	// **********************************************************
	// *                 MANAGEMENT TRANSITION                  *
	// **********************************************************
	
	// Transition from Stop to WarmUp
	
	IF "SM1".xBattOpenSt AND NOT "SM1".xStopAutomaintCmd        //Whit battery open and not automaintenance go to warmup state
	THEN
	    "SM1".xT81 := True;
	END_IF;
	
	// Reset Transition
	
	"SM1".xT32   := False;
	"SM1".xT43   := False;
	"SM1".xT52   := False;
	"SM1".xT72   := False;
	
END_FUNCTION

FUNCTION "SM1_S9_Fault" : Void
{ S7_Optimized_Access := 'TRUE' }
VERSION : 0.1

BEGIN
	// **********************************************************
	// *                   MANAGEMENT ACTION                    *
	// **********************************************************
	
	REGION State Machine Status
	    
	    "SM1".xSsBootSt      := False;
	    "SM1".xSsWarmUpSt    := False;
	    "SM1".xSsReadySt     := False;
	    "SM1".xSsStandBySt   := False;
	    "SM1".xSsRunSt       := False;
	    "SM1".xSsTestSt      := False;
	    "SM1".xSsAutoMaintSt := False;
	    "SM1".xSsStopSt      := False;
	    "SM1".xSsFaultSt     := True;
	    
	    "SM1".iCountSS := 9;
	    
	END_REGION
	
	"SM1".xPCSrunCmd := False;      //In fault state send stop command to the PCS
	
	REGION PCS enable Off
	    
	    IF "SM1".xPCSreadySt        //When the PCS are in ready take out the enable command to the PCS
	    THEN
	        "SM1".xPCSenbCmd := False;
	    END_IF;
	END_REGION
	
	REGION Command Open RMU and Battery
	    
	    IF "SM1".xPCSstopSt AND NOT "SM1".xVacPCS       //When we go in fault state have a possibility who the medium voltage is off
	    THEN
	        "SM1".xMVbreakerOpenCmd := True;        //If the medium voltage is off we need to open a MV breaker because otherwise after giving the open command to the battery,
	                                                //the PCS would switch off AND in this CASE you could NOT close the MV breaker anymore
	        IF "SM1".xMVbreakerOpenSt       //When the MV breaker are opened semd a open command to the battery
	        THEN
	            "SM1".xBattCloseCmd := False;
	        END_IF;
	    END_IF;
	    
	END_REGION
	
	REGION Command Open Battery
	    
	    IF "SM1".xPCSstopSt AND "SM1".xVacPCS       //If the medium voltage is on and PCS stopped send a open command to the battery
	    THEN
	        "SM1".xBattCloseCmd := False;
	    END_IF;
	    
	END_REGION
	
	
	// **********************************************************
	// *                 MANAGEMENT TRANSITION                  *
	// **********************************************************
	
	// Transition from Alarm to WarmUp
	
	IF NOT "SM1".xFltSt AND "SM1".xBattOpenSt       //Without faults and battery open return in warmup state
	THEN
	    "SM1".xT91 := True;
	    "SM1".xMVbreakerOpenCmd := False;
	END_IF;
	
	// Reset Transition
	
	"SM1".xT22   := False;
	"SM1".xT33   := False;
	"SM1".xT44   := False;
	"SM1".xT53   := False;
	"SM1".xT62   := False;
	"SM1".xT73   := False;
	
END_FUNCTION

FUNCTION "SM2_S1_Boot" : Void
{ S7_Optimized_Access := 'TRUE' }
VERSION : 0.1
   VAR_TEMP 
      xBoot_Ok : Bool;
      iT1 : S5Time;
   END_VAR


BEGIN
	// **********************************************************
	// *                   MANAGEMENT ACTION                    *
	// **********************************************************
	
	REGION State Machine Status
	    
	    "SM2".xSsBootSt      := True;
	    "SM2".xSsWarmUpSt    := False;
	    "SM2".xSsReadySt     := False;
	    "SM2".xSsStandBySt   := False;
	    "SM2".xSsRunSt       := False;
	    "SM2".xSsTestSt      := False;
	    "SM2".xSsAutoMaintSt := False;
	    "SM2".xSsStopSt      := False;
	    "SM2".xSsFaultSt     := False;
	    
	    "SM2".iCountSS := 1;
	    
	END_REGION
	
	REGION Wait PLC Status From Off to On
	    
	// When the PLC switch to Run after 5sec "xBootSt = True" and the transition "T1 = True"
	    
	#iT1 := S_ODT(
	    T_NO := 1,
	    S := "SM2".xRunPlcSt,
	    TV := S5T#5s,
	    Q => "SM2".xBootSt);
	END_REGION
	
	// **********************************************************
	// *                 MANAGEMENT TRANSITION                  *
	// **********************************************************
	
	// Transition from Boot to WarmUp
	
	IF "SM2".xBootSt
	THEN
	    "SM2".xT11 := True;
	    "SM2".xBootSt := False;
	END_IF;
	
END_FUNCTION

FUNCTION "SM2_S2_WarmUp" : Void
{ S7_Optimized_Access := 'TRUE' }
VERSION : 0.1
   VAR_TEMP 
      xWarmUpSt : Bool;
   END_VAR


BEGIN
	// **********************************************************
	// *                   MANAGEMENT ACTION                    *
	// **********************************************************
	
	REGION State Machine Status
	    
	    "SM2".xSsBootSt      := False;
	    "SM2".xSsWarmUpSt    := True;
	    "SM2".xSsReadySt     := False;
	    "SM2".xSsStandBySt   := False;
	    "SM2".xSsRunSt       := False;
	    "SM2".xSsTestSt      := False;
	    "SM2".xSsAutoMaintSt := False;
	    "SM2".xSsStopSt      := False;
	    "SM2".xSsFaultSt     := False;
	    
	    "SM2".iCountSS       := 2;
	    
	END_REGION
	
	REGION Activation
	    
	    "SM2".xCommCmd   := True;    //Enable all communication on the Power Island
	    "SM2".xAuxCmd    := True;    //Enable all auxiliary equipment on the Power Island
	    
	END_REGION
	
	REGION Activation Active
	    
	    IF "SM2".xAuxSt AND "SM2".xCommSt     //Check the feedback of communication and auxiliary on the Power Island
	    THEN
	        #xWarmUpSt := True;
	
	    END_IF;
	    
	END_REGION
	
	
	// **********************************************************
	// *                 MANAGEMENT TRANSITION                  *
	// **********************************************************
	
	// Transition from WarmUp to Ready
	
	IF #xWarmUpSt
	THEN
	    "SM2".xT21 := True;
	    #xWarmUpSt := False;
	END_IF;
	
	// Transition from WarmUp to Fault
	
	IF "SM2".xFltSt
	THEN
	    "SM2".xT22 := True;
	END_IF;
	
	// Reset Transition
	
	"SM2".xT11   := False;
	"SM2".xT81   := False;
	"SM2".xT91   := False;
	
END_FUNCTION

FUNCTION "SM2_S3_Ready" : Void
{ S7_Optimized_Access := 'TRUE' }
VERSION : 0.1
   VAR_TEMP 
      xSSysReadySt : Bool;
   END_VAR


BEGIN
	// **********************************************************
	// *                   MANAGEMENT ACTION                    *
	// **********************************************************
	
	REGION State Machine Status
	    
	    "SM2".xSsBootSt      := False;
	    "SM2".xSsWarmUpSt    := False;
	    "SM2".xSsReadySt     := True;
	    "SM2".xSsStandBySt   := False;
	    "SM2".xSsRunSt       := False;
	    "SM2".xSsTestSt      := False;
	    "SM2".xSsAutoMaintSt := False;
	    "SM2".xSsStopSt      := False;
	    "SM2".xSsFaultSt     := False;
	        
	    "SM2".iCountSS := 3;
	    
	END_REGION
	
	REGION Ready Condition
	    
	    IF "SM2".xReadyCondSt AND "SM2".xEnbSSysSt      //With ready condition and Subsystem enabled from HMI the subsystem is ready
	    THEN
	        #xSSysReadySt := True;
	    END_IF;
	    
	END_REGION
	
	REGION Command Battery Close
	    
	    IF #xSSysReadySt AND ("SM2".xStandByCmd OR "SM2".xRunCmd)       //With subsystem ready and standby or run command send close command to the battery
	    THEN
	        "SM2".xBattCloseCmd := True;
	    END_IF;
	    
	END_REGION
	
	REGION Command Enable PCS
	    
	    IF "SM2".xBattCloseSt AND "SM2".xMVbreakerCloseSt       //When the battery are closed and MV circuit breaker close send enable command to the PCS
	    THEN
	        "SM2".xPCSenbCmd := True;
	    END_IF;
	END_REGION
	
	
	// **********************************************************
	// *                 MANAGEMENT TRANSITION                  *
	// **********************************************************
	
	// Transition from Ready to StandBy
	
	IF "SM2".xBattCloseSt AND "SM2".xPCSreadySt     //With battery closed and PCS in ready condition go on standby state
	THEN
	    "SM2".xT31 := True;
	    #xSSysReadySt := False;
	END_IF;
	
	// Transition from Ready to Stop
	
	IF "SM2".xStopCmd AND False     //From ready status never go in stop state
	THEN
	    "SM2".xT32 := True;
	END_IF;
	
	// Transition from Ready to Fault
	
	IF "SM2".xFltSt     //With subsystem in fault go to the fault state
	THEN
	    "SM2".xT33 := True;
	END_IF;
	
	// Transition from Ready to Test
	
	IF "SM2".xTestCmd       //With test command from HMI go to the test state
	THEN
	    "SM2".xT34 := True;
	END_IF;
	
	// Reset Transition
	
	"SM2".xT21   := False;
	"SM2".xT61   := False;
	
END_FUNCTION

FUNCTION "SM2_S4_StandBy" : Void
{ S7_Optimized_Access := 'TRUE' }
VERSION : 0.1

BEGIN
	// **********************************************************
	// *                   MANAGEMENT ACTION                    *
	// **********************************************************
	
	REGION State Machine Status
	    
	    "SM2".xSsBootSt      := False;
	    "SM2".xSsWarmUpSt    := False;
	    "SM2".xSsReadySt     := False;
	    "SM2".xSsStandBySt   := True;
	    "SM2".xSsRunSt       := False;
	    "SM2".xSsTestSt      := False;
	    "SM2".xSsAutoMaintSt := False;
	    "SM2".xSsStopSt      := False;
	    "SM2".xSsFaultSt     := False;
	    
	    "SM2".iCountSS := 4;
	    
	END_REGION
	
	REGION Run Command
	    
	    IF "SM2".xRunCmd        //With run command send run command to the PCS
	    THEN
	        "SM2".xPCSrunCmd := True;
	    END_IF;
	    
	END_REGION
	
	
	// **********************************************************
	// *                 MANAGEMENT TRANSITION                  *
	// **********************************************************
	
	// Transition from StandBy to Run
	
	IF "SM2".xPCSrunSt AND "SM2".xRunCmd        //With PCS in run and the command on go to run state
	THEN
	    "SM2".xT41 := True;
	END_IF;
	
	// Transition from StandBy to AutoMaint
	
	IF "SM2".xAutomaintCmd      //With automaintenance command go to automaintenance state
	THEN
	    "SM2".xT42 := True;
	END_IF;
	
	// Transition from StandBy to Stop
	
	IF "SM2".xStopCmd OR NOT "SM2".xEnbSSysSt       //With stop command or subsystem not enabled go to stop state
	THEN
	    "SM2".xT43 := True;
	END_IF;
	
	// Transition from StandBy to Fault
	
	IF "SM2".xFltSt     //With subsystem in fault go to the fault state
	THEN
	    "SM2".xT44 := True;
	END_IF;
	
	// Reset Transition
	
	"SM2".xT31   := False;
	"SM2".xT51   := False;
	"SM2".xT71   := False;
	
END_FUNCTION

FUNCTION "SM2_S5_Run" : Void
{ S7_Optimized_Access := 'TRUE' }
VERSION : 0.1

BEGIN
	// **********************************************************
	// *                   MANAGEMENT ACTION                    *
	// **********************************************************
	
	REGION State Machine Status
	    
	    "SM2".xSsBootSt      := False;
	    "SM2".xSsWarmUpSt    := False;
	    "SM2".xSsReadySt     := False;
	    "SM2".xSsStandBySt   := False;
	    "SM2".xSsRunSt       := True;
	    "SM2".xSsTestSt      := False;
	    "SM2".xSsAutoMaintSt := False;
	    "SM2".xSsStopSt      := False;
	    "SM2".xSsFaultSt     := False;
	    
	    "SM2".iCountSS := 5;
	    
	END_REGION
	
	REGION StandBy Command
	    
	    IF "SM2".xStandByCmd        //With standby command send stop command to the PCS
	    THEN
	        "SM2".xPCSrunCmd := False;
	    END_IF;
	    
	END_REGION
	
	
	// **********************************************************
	// *                 MANAGEMENT TRANSITION                  *
	// **********************************************************
	
	// Transition from Run to StandBy
	
	IF "SM2".xStandByCmd AND "SM2".xPCSreadySt      //With standby command e PCS in ready return to standby state
	THEN
	    "SM2".xT51 := True;
	END_IF;
	
	// Transition from Run to Stop
	
	IF "SM2".xStopCmd OR NOT "SM2".xEnbSSysSt       //With stop command or subsystem not enabled go to stop state
	THEN
	    "SM2".xT52 := True;
	END_IF;
	
	// Transition from Run to Fault
	
	IF "SM2".xFltSt     //With subsystem in fault go to the fault state
	THEN
	    "SM2".xT53 := True;
	END_IF;
	
	// Reset Transition
	
	"SM2".xT41 := False;
	
END_FUNCTION

FUNCTION "SM2_S6_Test" : Void
{ S7_Optimized_Access := 'TRUE' }
VERSION : 0.1

BEGIN
	// **********************************************************
	// *                   MANAGEMENT ACTION                    *
	// **********************************************************
	
	REGION State Machine Status
	    
	    "SM2".xSsBootSt := False;
	    "SM2".xSsWarmUpSt := False;
	    "SM2".xSsReadySt := False;
	    "SM2".xSsStandBySt := False;
	    "SM2".xSsRunSt := False;
	    "SM2".xSsTestSt := True;
	    "SM2".xSsAutoMaintSt := False;
	    "SM2".xSsStopSt := False;
	    "SM2".xSsFaultSt := False;
	    
	    "SM2".iCountSS := 6;
	    
	END_REGION
	
	"SM2".xPCSrunCmd := False;      //All command in this state are not necessary but only for safety
	
	REGION PCS Enable Off
	    
	    IF "SM2".xPCSreadySt
	    THEN
	        "SM2".xPCSenbCmd := False;
	    END_IF;
	END_REGION
	
	REGION Command Open Battery
	    
	    IF "SM2".xPCSstopSt
	    THEN
	        "SM2".xBattCloseCmd := False;
	    END_IF;
	END_REGION
	
	
	// **********************************************************
	// *                 MANAGEMENT TRANSITION                  *
	// **********************************************************
	
	// Transition from Test to Ready
	
	IF NOT "SM2".xTestCmd       //Without test command return to ready state
	THEN
	    "SM2".xT61 := True;
	END_IF;
	
	// Transition from Test to Fault
	
	IF "SM2".xFltSt     //With subsystem in fault go to the fault state
	THEN
	    "SM2".xT62 := True;
	END_IF;
	
	// Reset Transition
	
	"SM2".xT34 := False;
	
END_FUNCTION

FUNCTION "SM2_S7_AutoMaint" : Void
{ S7_Optimized_Access := 'TRUE' }
VERSION : 0.1

BEGIN
	// **********************************************************
	// *                   MANAGEMENT ACTION                    *
	// **********************************************************
	
	REGION State Machine Status
	    
	    "SM2".xSsBootSt      := False;
	    "SM2".xSsWarmUpSt    := False;
	    "SM2".xSsReadySt     := False;
	    "SM2".xSsStandBySt   := False;
	    "SM2".xSsRunSt       := False;
	    "SM2".xSsTestSt      := False;
	    "SM2".xSsAutoMaintSt := True;
	    "SM2".xSsStopSt      := False;
	    "SM2".xSsFaultSt     := False;
	    
	    "SM2".iCountSS := 7;
	    
	END_REGION
	
	REGION Autocharge Bank
	    
	    "SM2".xPCSrunCmd := True;       //In automaintenance state send run command to the PCS
	    
	    IF "SM2".xPCSrunSt      //When PCS are in run read the active power reference from HMI
	    THEN
	        "SM2".rPacAutomRef := "HMI".rPacAutomRef;
	    END_IF;
	    
	END_REGION
	
	
	// **********************************************************
	// *                 MANAGEMENT TRANSITION                  *
	// **********************************************************
	
	// Transition from AutoMaint to StandBy
	
	IF "SM2".xAutomaintSt       //Without automaintenance command from battery return to standby state
	THEN
	    "SM2".xT71 := True;
	END_IF;
	
	// Transition from AutoMaint to Stop
	
	IF "SM2".xStopCmd       //With stop command go to stop state
	THEN
	    "SM2".xT72 := True;
	END_IF;
	
	// Transition from AutoMaint to Fault
	
	IF "SM2".xFltSt     //With subsystem in fault go to the fault state
	THEN
	    "SM2".xT73 := True;
	END_IF;
	
	// Reset Transition
	
	"SM2".xT42    := False;
	
END_FUNCTION

FUNCTION "SM2_S8_Stop" : Void
{ S7_Optimized_Access := 'TRUE' }
VERSION : 0.1

BEGIN
	// **********************************************************
	// *                   MANAGEMENT ACTION                    *
	// **********************************************************
	
	REGION State Machine Status
	    
	    "SM2".xSsBootSt      := False;
	    "SM2".xSsWarmUpSt    := False;
	    "SM2".xSsReadySt     := False;
	    "SM2".xSsStandBySt   := False;
	    "SM2".xSsRunSt       := False;
	    "SM2".xSsTestSt      := False;
	    "SM2".xSsAutoMaintSt := False;
	    "SM2".xSsStopSt      := True;
	    "SM2".xSsFaultSt     := False;
	    
	    "SM2".iCountSS := 8;
	    
	END_REGION
	
	"SM2".xPCSrunCmd := False;      //In stop state send stop command to the PCS
	
	REGION PCS Enable Off
	    
	    IF "SM2".xPCSreadySt        //When the PCS are in ready take out the enable command to the PCS
	    THEN
	        "SM2".xPCSenbCmd := False;
	    END_IF;
	END_REGION
	
	REGION Command Open Battery
	    
	    IF "SM2".xPCSstopSt     //When the PCS are in stop send open command to the battery
	    THEN
	        "SM2".xBattCloseCmd := False;
	    END_IF;
	END_REGION
	
	
	// **********************************************************
	// *                 MANAGEMENT TRANSITION                  *
	// **********************************************************
	
	// Transition from Stop to WarmUp
	
	IF "SM2".xBattOpenSt AND NOT "SM2".xStopAutomaintCmd        //Whit battery open and not automaintenance go to warmup state
	THEN
	    "SM2".xT81 := True;
	END_IF;
	
	// Reset Transition
	
	"SM2".xT32   := False;
	"SM2".xT43   := False;
	"SM2".xT52   := False;
	"SM2".xT72   := False;
	
END_FUNCTION

FUNCTION "SM2_S9_Fault" : Void
{ S7_Optimized_Access := 'TRUE' }
VERSION : 0.1

BEGIN
	// **********************************************************
	// *                   MANAGEMENT ACTION                    *
	// **********************************************************
	
	REGION State Machine Status
	    
	    "SM2".xSsBootSt      := False;
	    "SM2".xSsWarmUpSt    := False;
	    "SM2".xSsReadySt     := False;
	    "SM2".xSsStandBySt   := False;
	    "SM2".xSsRunSt       := False;
	    "SM2".xSsTestSt      := False;
	    "SM2".xSsAutoMaintSt := False;
	    "SM2".xSsStopSt      := False;
	    "SM2".xSsFaultSt     := True;
	    
	    "SM2".iCountSS := 9;
	    
	END_REGION
	
	"SM2".xPCSrunCmd := False;      //In fault state send stop command to the PCS
	
	REGION PCS Enable Off
	    
	    IF "SM2".xPCSreadySt        //When the PCS are in ready take out the enable command to the PCS
	    THEN
	        "SM2".xPCSenbCmd := False;
	    END_IF;
	END_REGION
	
	REGION Command Open RMU and Battery
	    
	    IF "SM2".xPCSstopSt AND NOT "SM2".xVacPCS       //When we go in fault state have a possibility who the medium voltage is off
	    THEN
	        "SM2".xMVbreakerOpenCmd := True;        //If the medium voltage is off we need to open a MV breaker because otherwise after giving the open command to the battery,
	                                                //the PCS would switch off AND in this CASE you could NOT close the MV breaker anymore        
	        IF "SM2".xMVbreakerOpenSt       //When the MV breaker are opened semd a open command to the battery
	        THEN
	            "SM2".xBattCloseCmd := False;
	        END_IF;
	    END_IF;
	    
	END_REGION
	
	REGION Command Open Battery
	    
	    IF "SM2".xPCSstopSt AND "SM2".xVacPCS       //If the medium voltage is on and PCS stopped send a open command to the battery
	    THEN
	        "SM2".xBattCloseCmd := False;
	    END_IF;
	    
	END_REGION
	
	
	// **********************************************************
	// *                 MANAGEMENT TRANSITION                  *
	// **********************************************************
	
	// Transition from Alarm to WarmUp
	
	IF NOT "SM2".xFltSt AND "SM2".xBattOpenSt       //Without faults and battery open return in warmup state
	THEN
	    "SM2".xT91 := True;
	    "SM2".xMVbreakerOpenCmd := False;
	END_IF;
	
	// Reset Transition
	
	"SM2".xT22   := False;
	"SM2".xT33   := False;
	"SM2".xT44   := False;
	"SM2".xT53   := False;
	"SM2".xT62   := False;
	"SM2".xT73   := False;
	
END_FUNCTION

FUNCTION "PE_InvFlt_1" : Void
{ S7_Optimized_Access := 'TRUE' }
VERSION : 0.1
   VAR_INPUT 
      iInput : Int;
      xReset : Bool;
   END_VAR

   VAR_OUTPUT 
      wOut : Word;
   END_VAR

   VAR_TEMP 
      iCounter : Int;
   END_VAR

   VAR CONSTANT 
      iStart : Int := 1;
      iEnd : Int := 393;
   END_VAR


BEGIN
	FOR #iCounter := 1 TO #iEnd DO
	    // Statement section FOR
	    ;
	END_FOR;
	
	
	
END_FUNCTION

FUNCTION "PE_R_Block" : Void
{ S7_Optimized_Access := 'TRUE' }
VERSION : 0.1
   VAR_INPUT 
      Input_Data : Array[1..125] of Word;
   END_VAR

   VAR_OUTPUT 
      Output_Data : "R_PE";
   END_VAR

   VAR_TEMP 
      "DWord" : DWord;
   END_VAR


BEGIN
	REGION
	    // 2022/02/16
	END_REGION
	
	REGION
	    
	    #Output_Data.rPacMeas       := INT_TO_REAL(WORD_TO_INT(#Input_Data[1]));
	    #Output_Data.rQacMeas       := INT_TO_REAL(WORD_TO_INT(#Input_Data[2]));
	    #Output_Data.rSacMeas       := INT_TO_REAL(WORD_TO_INT(#Input_Data[3]));
	    #Output_Data.rPFmeas        := INT_TO_REAL(WORD_TO_INT(#Input_Data[4]))/1000.0;
	    #Output_Data.rFrMeas        := INT_TO_REAL(WORD_TO_INT(#Input_Data[5]))/100.0;
	    
	    #Output_Data.rVrsMeas       := INT_TO_REAL(WORD_TO_INT(#Input_Data[6]));
	    #Output_Data.rVstMeas       := INT_TO_REAL(WORD_TO_INT(#Input_Data[7]));
	    #Output_Data.rVtrMeas       := INT_TO_REAL(WORD_TO_INT(#Input_Data[8]));
	    #Output_Data.rIrMeas        := INT_TO_REAL(WORD_TO_INT(#Input_Data[9]));
	    #Output_Data.rIsMeas        := INT_TO_REAL(WORD_TO_INT(#Input_Data[10]));
	    #Output_Data.rItMeas        := INT_TO_REAL(WORD_TO_INT(#Input_Data[11]));
	     
	    #Output_Data.rPdcMeas       := INT_TO_REAL(WORD_TO_INT(#Input_Data[12]));
	    #Output_Data.rIdcMeas       := INT_TO_REAL(WORD_TO_INT(#Input_Data[13]));
	    
	    #Output_Data.iImonDc1St     := WORD_TO_INT(#Input_Data[14]);
	    
	    #Output_Data.iImonAcSt      := WORD_TO_INT(#Input_Data[15]);
	    
	    #Output_Data.iCodeFlt       := WORD_TO_INT(#Input_Data[16]);
	    #Output_Data.iCodeWarn      := WORD_TO_INT(#Input_Data[17]);
	    
	    #Output_Data.iCodeSt        := WORD_TO_INT(#Input_Data[18]);
	    #Output_Data.xInvOffSt      := #Output_Data.iCodeSt = 2;
	    #Output_Data.xInvStandBySt  := #Output_Data.iCodeSt = 14;
	    #Output_Data.xInvReadySt    := #Output_Data.iCodeSt = 4;
	    #Output_Data.xInvPrOnSt     := #Output_Data.iCodeSt = 17;
	    #Output_Data.xInvRunSt      := #Output_Data.iCodeSt = 6;
	    #Output_Data.xInvStopSt     := #Output_Data.iCodeSt = 7;
	    #Output_Data.xInvFltSt      := #Output_Data.iCodeSt = 9;
	    
	    #Output_Data.rTmodAcMeas    := INT_TO_REAL(WORD_TO_INT(#Input_Data[19]));
	    #Output_Data.rTigbtMaxMeas  := INT_TO_REAL(WORD_TO_INT(#Input_Data[20]));
	    #Output_Data.rTmodMaxMeas   := INT_TO_REAL(WORD_TO_INT(#Input_Data[21]));
	    
	    #Output_Data.wDIboardSt     := #Input_Data[22];
	    #Output_Data.wDOboardSt     := #Input_Data[23];
	    
	    #Output_Data.rTmodAcInMeas      := INT_TO_REAL(WORD_TO_INT(#Input_Data[24]))/10.0;
	    #Output_Data.iFltModId          := WORD_TO_INT(#Input_Data[25]);
	    #Output_Data.rRHintMeas         := INT_TO_REAL(WORD_TO_INT(#Input_Data[26]));
	    #Output_Data.rVaux1Meas         := INT_TO_REAL(WORD_TO_INT(#Input_Data[27]))/100.0;
	    #Output_Data.rVaux2Meas         := INT_TO_REAL(WORD_TO_INT(#Input_Data[28]))/100.0;
	    
	    #Output_Data.rPacAvlLim  := INT_TO_REAL(WORD_TO_INT(#Input_Data[29]))/1000.0;
	    #Output_Data.rQacAvlLim  := INT_TO_REAL(WORD_TO_INT(#Input_Data[30]))/1000.0;
	    
	    #Output_Data.wDUchanSel     := #Input_Data[31];
	    #Output_Data.wDUchanSt      := #Input_Data[42];
	    
	    #Output_Data.rVdcBus1Meas   := INT_TO_REAL(WORD_TO_INT(#Input_Data[32]));
	    #Output_Data.rVdcBus2Meas   := INT_TO_REAL(WORD_TO_INT(#Input_Data[33]));
	    #Output_Data.rIdcBus1Meas   := INT_TO_REAL(WORD_TO_INT(#Input_Data[34]));
	    #Output_Data.rIdcBus2Meas   := INT_TO_REAL(WORD_TO_INT(#Input_Data[35]));
	    #Output_Data.rIRFIcapRef    := INT_TO_REAL(WORD_TO_INT(#Input_Data[36]))/10.0;
	    
	    #Output_Data.rPavlChaBus1   := INT_TO_REAL(WORD_TO_INT(#Input_Data[37]))/100.0;
	    #Output_Data.rPavlDschBus1 := INT_TO_REAL(WORD_TO_INT(#Input_Data[38]))/100.0;
	    #Output_Data.rPavlChaBus2   := INT_TO_REAL(WORD_TO_INT(#Input_Data[39]))/100.0;
	    #Output_Data.rPavlDschBus2 := INT_TO_REAL(WORD_TO_INT(#Input_Data[40]))/100.0;
	    
	    #Output_Data.iImonDc2St     := WORD_TO_INT(#Input_Data[41]);
	    
	    #Output_Data.wMod1St        := WORD_TO_INT(#Input_Data[43]);
	    #Output_Data.xMod1StopSt    := #Output_Data.wMod1St = 1;
	    #Output_Data.xMod1ReadySt   := #Output_Data.wMod1St = 3;
	    #Output_Data.xMod1MainAcSt  := #Output_Data.wMod1St = 5;
	    #Output_Data.xMod1RunSt     := #Output_Data.wMod1St = 7;
	    #Output_Data.xMod1FltSt     := #Output_Data.wMod1St = 20;
	    
	    #Output_Data.rMod1PacMeas   := INT_TO_REAL(WORD_TO_INT(#Input_Data[44]))/10.0;
	    #Output_Data.rMod1QacMeas   := INT_TO_REAL(WORD_TO_INT(#Input_Data[45]))/10.0;
	    
	    #Output_Data.wMod1IOSt          := #Input_Data[46];
	    #Output_Data.xMod1ThermLCLst    := #Output_Data.wMod1IOSt.%X6;
	    #Output_Data.xMod1FanSt         := #Output_Data.wMod1IOSt.%X7;
	    #Output_Data.xMod1AcMainSt      := #Output_Data.wMod1IOSt.%X8;
	    #Output_Data.xMod1AcSoftChaSt   := #Output_Data.wMod1IOSt.%X9;
	    #Output_Data.xMod1LCLst         := #Output_Data.wMod1IOSt.%X10;
	    #Output_Data.xMod1DcSwitchSt    := #Output_Data.wMod1IOSt.%X11;
	    
	    #Output_Data.rMod1TempR1Meas    := INT_TO_REAL(WORD_TO_INT(#Input_Data[47]));
	    #Output_Data.rMod1TempR2Meas    := INT_TO_REAL(WORD_TO_INT(#Input_Data[48]));
	    #Output_Data.rMod1TempR3Meas    := INT_TO_REAL(WORD_TO_INT(#Input_Data[49]));
	    #Output_Data.rMod1TempS1Meas    := INT_TO_REAL(WORD_TO_INT(#Input_Data[50]));
	    #Output_Data.rMod1TempS2Meas    := INT_TO_REAL(WORD_TO_INT(#Input_Data[51]));
	    #Output_Data.rMod1TempS3Meas    := INT_TO_REAL(WORD_TO_INT(#Input_Data[52]));
	    #Output_Data.rMod1TempT1Meas    := INT_TO_REAL(WORD_TO_INT(#Input_Data[53]));
	    #Output_Data.rMod1TempT2Meas    := INT_TO_REAL(WORD_TO_INT(#Input_Data[54]));
	    #Output_Data.rMod1TempT3Meas    := INT_TO_REAL(WORD_TO_INT(#Input_Data[55]));
	    
	    #Output_Data.wMod2St        := WORD_TO_INT(#Input_Data[56]);
	    #Output_Data.xMod2StopSt    := #Output_Data.wMod2St = 1;
	    #Output_Data.xMod2ReadySt   := #Output_Data.wMod2St = 3;
	    #Output_Data.xMod2MainAcSt  := #Output_Data.wMod2St = 5;
	    #Output_Data.xMod2RunSt     := #Output_Data.wMod2St = 7;
	    #Output_Data.xMod2FltSt     := #Output_Data.wMod2St = 20;
	    
	    #Output_Data.rMod2PacMeas   := INT_TO_REAL(WORD_TO_INT(#Input_Data[57]))/10.0;
	    #Output_Data.rMod2QacMeas   := INT_TO_REAL(WORD_TO_INT(#Input_Data[58]))/10.0;
	    
	    #Output_Data.wMod2IOSt          := #Input_Data[59];
	    #Output_Data.xMod2ThermLCLst    := #Output_Data.wMod2IOSt.%X6;
	    #Output_Data.xMod2FanSt         := #Output_Data.wMod2IOSt.%X7;
	    #Output_Data.xMod2AcMainSt      := #Output_Data.wMod2IOSt.%X8;
	    #Output_Data.xMod2AcSoftChaSt   := #Output_Data.wMod2IOSt.%X9;
	    #Output_Data.xMod2LCLst         := #Output_Data.wMod2IOSt.%X10;
	    #Output_Data.xMod2DcSwitchSt    := #Output_Data.wMod2IOSt.%X11;
	    
	    #Output_Data.rMod2TempR1Meas    := INT_TO_REAL(WORD_TO_INT(#Input_Data[60]));
	    #Output_Data.rMod2TempR2Meas    := INT_TO_REAL(WORD_TO_INT(#Input_Data[61]));
	    #Output_Data.rMod2TempR3Meas    := INT_TO_REAL(WORD_TO_INT(#Input_Data[62]));
	    #Output_Data.rMod2TempS1Meas    := INT_TO_REAL(WORD_TO_INT(#Input_Data[63]));
	    #Output_Data.rMod2TempS2Meas    := INT_TO_REAL(WORD_TO_INT(#Input_Data[64]));
	    #Output_Data.rMod2TempS3Meas    := INT_TO_REAL(WORD_TO_INT(#Input_Data[65]));
	    #Output_Data.rMod2TempT1Meas    := INT_TO_REAL(WORD_TO_INT(#Input_Data[66]));
	    #Output_Data.rMod2TempT2Meas    := INT_TO_REAL(WORD_TO_INT(#Input_Data[67]));
	    #Output_Data.rMod2TempT3Meas    := INT_TO_REAL(WORD_TO_INT(#Input_Data[68]));
	    
	    #Output_Data.wMod3St        := WORD_TO_INT(#Input_Data[69]);
	    #Output_Data.xMod3StopSt    := #Output_Data.wMod3St = 1;
	    #Output_Data.xMod3ReadySt   := #Output_Data.wMod3St = 3;
	    #Output_Data.xMod3MainAcSt  := #Output_Data.wMod3St = 5;
	    #Output_Data.xMod3RunSt     := #Output_Data.wMod3St = 7;
	    #Output_Data.xMod3FltSt     := #Output_Data.wMod3St = 20;
	    
	    #Output_Data.rMod3PacMeas   := INT_TO_REAL(WORD_TO_INT(#Input_Data[70]))/10.0;
	    #Output_Data.rMod3QacMeas   := INT_TO_REAL(WORD_TO_INT(#Input_Data[71]))/10.0;
	    
	    #Output_Data.wMod3IOSt          := #Input_Data[72];
	    #Output_Data.xMod3ThermLCLst    := #Output_Data.wMod3IOSt.%X6;
	    #Output_Data.xMod3FanSt         := #Output_Data.wMod3IOSt.%X7;
	    #Output_Data.xMod3AcMainSt      := #Output_Data.wMod3IOSt.%X8;
	    #Output_Data.xMod3AcSoftChaSt   := #Output_Data.wMod3IOSt.%X9;
	    #Output_Data.xMod3LCLst         := #Output_Data.wMod3IOSt.%X10;
	    #Output_Data.xMod3DcSwitchSt    := #Output_Data.wMod3IOSt.%X11;
	    
	    #Output_Data.rMod3TempR1Meas    := INT_TO_REAL(WORD_TO_INT(#Input_Data[73]));
	    #Output_Data.rMod3TempR2Meas    := INT_TO_REAL(WORD_TO_INT(#Input_Data[74]));
	    #Output_Data.rMod3TempR3Meas    := INT_TO_REAL(WORD_TO_INT(#Input_Data[75]));
	    #Output_Data.rMod3TempS1Meas    := INT_TO_REAL(WORD_TO_INT(#Input_Data[76]));
	    #Output_Data.rMod3TempS2Meas    := INT_TO_REAL(WORD_TO_INT(#Input_Data[77]));
	    #Output_Data.rMod3TempS3Meas    := INT_TO_REAL(WORD_TO_INT(#Input_Data[78]));
	    #Output_Data.rMod3TempT1Meas    := INT_TO_REAL(WORD_TO_INT(#Input_Data[79]));
	    #Output_Data.rMod3TempT2Meas    := INT_TO_REAL(WORD_TO_INT(#Input_Data[80]));
	    #Output_Data.rMod3TempT3Meas    := INT_TO_REAL(WORD_TO_INT(#Input_Data[81]));
	    
	    #Output_Data.wMod4St        := WORD_TO_INT(#Input_Data[82]);
	    #Output_Data.xMod4StopSt    := #Output_Data.wMod4St = 1;
	    #Output_Data.xMod4ReadySt   := #Output_Data.wMod4St = 3;
	    #Output_Data.xMod4MainAcSt  := #Output_Data.wMod4St = 5;
	    #Output_Data.xMod4RunSt     := #Output_Data.wMod4St = 7;
	    #Output_Data.xMod4FltSt     := #Output_Data.wMod4St = 20;
	    
	    #Output_Data.rMod4PacMeas   := INT_TO_REAL(WORD_TO_INT(#Input_Data[83]))/10.0;
	    #Output_Data.rMod4QacMeas   := INT_TO_REAL(WORD_TO_INT(#Input_Data[84]))/10.0;
	    
	    #Output_Data.wMod4IOSt          := #Input_Data[85];
	    #Output_Data.xMod4ThermLCLst    := #Output_Data.wMod4IOSt.%X6;
	    #Output_Data.xMod4FanSt         := #Output_Data.wMod4IOSt.%X7;
	    #Output_Data.xMod4AcMainSt      := #Output_Data.wMod4IOSt.%X8;
	    #Output_Data.xMod4AcSoftChaSt   := #Output_Data.wMod4IOSt.%X9;
	    #Output_Data.xMod4LCLst         := #Output_Data.wMod4IOSt.%X10;
	    #Output_Data.xMod4DcSwitchSt    := #Output_Data.wMod4IOSt.%X11;
	    
	    #Output_Data.rMod4TempR1Meas    := INT_TO_REAL(WORD_TO_INT(#Input_Data[86]));
	    #Output_Data.rMod4TempR2Meas    := INT_TO_REAL(WORD_TO_INT(#Input_Data[87]));
	    #Output_Data.rMod4TempR3Meas    := INT_TO_REAL(WORD_TO_INT(#Input_Data[88]));
	    #Output_Data.rMod4TempS1Meas    := INT_TO_REAL(WORD_TO_INT(#Input_Data[89]));
	    #Output_Data.rMod4TempS2Meas    := INT_TO_REAL(WORD_TO_INT(#Input_Data[90]));
	    #Output_Data.rMod4TempS3Meas    := INT_TO_REAL(WORD_TO_INT(#Input_Data[91]));
	    #Output_Data.rMod4TempT1Meas    := INT_TO_REAL(WORD_TO_INT(#Input_Data[92]));
	    #Output_Data.rMod4TempT2Meas    := INT_TO_REAL(WORD_TO_INT(#Input_Data[93]));
	    #Output_Data.rMod4TempT3Meas    := INT_TO_REAL(WORD_TO_INT(#Input_Data[94]));
	    
	    #Output_Data.wMod5St        := WORD_TO_INT(#Input_Data[95]);
	    #Output_Data.xMod5StopSt    := #Output_Data.wMod5St = 1;
	    #Output_Data.xMod5ReadySt   := #Output_Data.wMod5St = 3;
	    #Output_Data.xMod5MainAcSt  := #Output_Data.wMod5St = 5;
	    #Output_Data.xMod5RunSt     := #Output_Data.wMod5St = 7;
	    #Output_Data.xMod5FltSt     := #Output_Data.wMod5St = 20;
	    
	    #Output_Data.rMod5PacMeas   := INT_TO_REAL(WORD_TO_INT(#Input_Data[96]))/10.0;
	    #Output_Data.rMod5QacMeas   := INT_TO_REAL(WORD_TO_INT(#Input_Data[97]))/10.0;
	    
	    #Output_Data.wMod5IOSt          := #Input_Data[98];
	    #Output_Data.xMod5ThermLCLst    := #Output_Data.wMod5IOSt.%X6;
	    #Output_Data.xMod5FanSt         := #Output_Data.wMod5IOSt.%X7;
	    #Output_Data.xMod5AcMainSt      := #Output_Data.wMod5IOSt.%X8;
	    #Output_Data.xMod5AcSoftChaSt   := #Output_Data.wMod5IOSt.%X9;
	    #Output_Data.xMod5LCLst         := #Output_Data.wMod5IOSt.%X10;
	    #Output_Data.xMod5DcSwitchSt    := #Output_Data.wMod5IOSt.%X11;
	    
	    #Output_Data.rMod5TempR1Meas    := INT_TO_REAL(WORD_TO_INT(#Input_Data[99]));
	    #Output_Data.rMod5TempR2Meas    := INT_TO_REAL(WORD_TO_INT(#Input_Data[100]));
	    #Output_Data.rMod5TempR3Meas    := INT_TO_REAL(WORD_TO_INT(#Input_Data[101]));
	    #Output_Data.rMod5TempS1Meas    := INT_TO_REAL(WORD_TO_INT(#Input_Data[102]));
	    #Output_Data.rMod5TempS2Meas    := INT_TO_REAL(WORD_TO_INT(#Input_Data[103]));
	    #Output_Data.rMod5TempS3Meas    := INT_TO_REAL(WORD_TO_INT(#Input_Data[104]));
	    #Output_Data.rMod5TempT1Meas    := INT_TO_REAL(WORD_TO_INT(#Input_Data[105]));
	    #Output_Data.rMod5TempT2Meas    := INT_TO_REAL(WORD_TO_INT(#Input_Data[106]));
	    #Output_Data.rMod5TempT3Meas    := INT_TO_REAL(WORD_TO_INT(#Input_Data[107]));
	    
	    #Output_Data.wMod6St        := WORD_TO_INT(#Input_Data[108]);
	    #Output_Data.xMod6StopSt    := #Output_Data.wMod6St = 1;
	    #Output_Data.xMod6ReadySt   := #Output_Data.wMod6St = 3;
	    #Output_Data.xMod6MainAcSt  := #Output_Data.wMod6St = 5;
	    #Output_Data.xMod6RunSt     := #Output_Data.wMod6St = 7;
	    #Output_Data.xMod6FltSt     := #Output_Data.wMod6St = 20;
	    
	    #Output_Data.rMod6PacMeas   := INT_TO_REAL(WORD_TO_INT(#Input_Data[109]))/10.0;
	    #Output_Data.rMod6QacMeas   := INT_TO_REAL(WORD_TO_INT(#Input_Data[110]))/10.0;
	    
	    #Output_Data.wMod6IOSt          := #Input_Data[111];
	    #Output_Data.xMod6ThermLCLst    := #Output_Data.wMod6IOSt.%X6;
	    #Output_Data.xMod6FanSt         := #Output_Data.wMod6IOSt.%X7;
	    #Output_Data.xMod6AcMainSt      := #Output_Data.wMod6IOSt.%X8;
	    #Output_Data.xMod6AcSoftChaSt   := #Output_Data.wMod6IOSt.%X9;
	    #Output_Data.xMod6LCLst         := #Output_Data.wMod6IOSt.%X10;
	    #Output_Data.xMod6DcSwitchSt    := #Output_Data.wMod6IOSt.%X11;
	    
	    #Output_Data.rMod6TempR1Meas    := INT_TO_REAL(WORD_TO_INT(#Input_Data[112]));
	    #Output_Data.rMod6TempR2Meas    := INT_TO_REAL(WORD_TO_INT(#Input_Data[113]));
	    #Output_Data.rMod6TempR3Meas    := INT_TO_REAL(WORD_TO_INT(#Input_Data[114]));
	    #Output_Data.rMod6TempS1Meas    := INT_TO_REAL(WORD_TO_INT(#Input_Data[115]));
	    #Output_Data.rMod6TempS2Meas    := INT_TO_REAL(WORD_TO_INT(#Input_Data[116]));
	    #Output_Data.rMod6TempS3Meas    := INT_TO_REAL(WORD_TO_INT(#Input_Data[117]));
	    #Output_Data.rMod6TempT1Meas    := INT_TO_REAL(WORD_TO_INT(#Input_Data[118]));
	    #Output_Data.rMod6TempT2Meas    := INT_TO_REAL(WORD_TO_INT(#Input_Data[119]));
	    #Output_Data.rMod6TempT3Meas    := INT_TO_REAL(WORD_TO_INT(#Input_Data[120]));
	    
	END_REGION
END_FUNCTION

FUNCTION "PE_W_Block1_old" : Void
{ S7_Optimized_Access := 'TRUE' }
VERSION : 0.1
   VAR_INPUT 
      In_Data : "W_PE";   // pcs
   END_VAR

   VAR_OUTPUT 
      Out_Data : Array[1..125] of Word;
   END_VAR


BEGIN
	REGION
	    #Out_Data[1] := #In_Data."wUserPswIns";
	END_REGION
END_FUNCTION

FUNCTION "PE_W_Block2_old" : Void
{ S7_Optimized_Access := 'TRUE' }
VERSION : 0.1
   VAR_INPUT 
      In_Data : "W_PE";   // udt. Samsung Data rack 1
   END_VAR

   VAR_OUTPUT 
      Out_Data : Array[1..125] of Word;
   END_VAR


BEGIN
	//27/03/2023
	
	REGION
	    #Out_Data[1]    := INT_TO_WORD(#In_Data."iModePctrlCmd");
	    #Out_Data[2]    := INT_TO_WORD(#In_Data."iModeQctrlCmd");
	END_REGION
END_FUNCTION

FUNCTION "PE_W_Block3_old" : Void
{ S7_Optimized_Access := 'TRUE' }
VERSION : 0.1
   VAR_INPUT 
      In_Data : Real;
   END_VAR

   VAR_OUTPUT 
      Out_Data : Array[1..125] of Word;
   END_VAR


BEGIN
	
	REGION
	    #Out_Data[1] := INT_TO_WORD(REAL_TO_INT(#In_Data * 100.0));
	END_REGION
END_FUNCTION

DATA_BLOCK "LPNDR_ET200"   // DB402
AUTHOR : SIOS
FAMILY : LPNDR
VERSION : 2.0
// stored: AutoNumber false, DBAccessibleFromOPCUA true, DBAccessibleFromWebserver true, InstanceOfName LPNDR_ReadGlobalInfo, InstanceOfType FB
"LPNDR_ReadGlobalInfo"
   // VAR_INPUT
   //    execute : Bool;
   //    hwId : HW_IO;
   // END_VAR
   // VAR_OUTPUT
   //    done { ExternalWritable := 'False'} : Bool;
   //    busy { ExternalWritable := 'False'} : Bool;
   //    error { ExternalWritable := 'False'} : Bool;
   //    status { ExternalWritable := 'False'} : Word;
   //    InterfaceInformation : "LPNDR_typeInterfaceInformation";
   //    PortInformation : Array[1..52] of "LPNDR_typePortInformation";
   //    PortLinkState : Array[1..52] of "LPNDR_typePortLinkState";
   //    PortStatistic : Array[1..52] of "LPNDR_typePortStatistic";
   //    diagnostics { ExternalWritable := 'False'} : "typeDiagnostics";
   // END_VAR
   // VAR
   //    statExecuteOld { ExternalAccessible := 'False'; ExternalVisible := 'False'; ExternalWritable := 'False'} : Bool;
   //    statDone { ExternalAccessible := 'False'; ExternalVisible := 'False'; ExternalWritable := 'False'} : Bool;
   //    statBusy { ExternalAccessible := 'False'; ExternalVisible := 'False'; ExternalWritable := 'False'} : Bool;
   //    statError { ExternalAccessible := 'False'; ExternalVisible := 'False'; ExternalWritable := 'False'} : Bool;
   //    statStatus { ExternalAccessible := 'False'; ExternalVisible := 'False'; ExternalWritable := 'False'} : Word;
   //    statSubfunctionStatus { ExternalAccessible := 'False'; ExternalVisible := 'False'; ExternalWritable := 'False'} : Word;
   //    statFBErrorState { ExternalAccessible := 'False'; ExternalVisible := 'False'; ExternalWritable := 'False'} : DInt;
   //    statFBState { ExternalAccessible := 'False'; ExternalVisible := 'False'; ExternalWritable := 'False'} : DInt;
   //    statEmptyDiagnostics { ExternalAccessible := 'False'; ExternalVisible := 'False'; ExternalWritable := 'False'} : "typeDiagnostics";
   //    InstReadRecord { S7_SetPoint := 'True'} : RDREC;
   //    statReadRecordLength : UInt;
   //    statReadRecordRequest : Bool;
   //    statPDInterfaceMrpDataReal : UInt;
   //    statPDPortMrpDataReal : UInt;
   //    statPDInterfaceDataReal : UInt;
   //    statPDPortDataReal : UInt;
   //    statPDPortStatistic : UInt;
   //    statUnknown : UInt;
   //    statInterfaceInfoReset : "LPNDR_typeInterfaceInformation";
   //    statPortInfoReset { S7_SetPoint := 'True'} : "LPNDR_typePortInformation";
   //    statPortLinkStateReset { S7_SetPoint := 'True'} : "LPNDR_typePortLinkState";
   //    statPortStatisticReset { S7_SetPoint := 'True'} : "LPNDR_typePortStatistic";
   //    statReadRecord { S7_SetPoint := 'True'} : Array[0..4175] of Byte;
   // END_VAR
BEGIN
END_DATA_BLOCK

DATA_BLOCK "LPNDR_PEMS"   // DB401
AUTHOR : SIOS
FAMILY : LPNDR
VERSION : 2.0
// stored: AutoNumber false, DBAccessibleFromOPCUA true, DBAccessibleFromWebserver true, InstanceOfName LPNDR_ReadGlobalInfo, InstanceOfType FB
"LPNDR_ReadGlobalInfo"
   // VAR_INPUT
   //    execute : Bool;
   //    hwId : HW_IO;
   // END_VAR
   // VAR_OUTPUT
   //    done { ExternalWritable := 'False'} : Bool;
   //    busy { ExternalWritable := 'False'} : Bool;
   //    error { ExternalWritable := 'False'} : Bool;
   //    status { ExternalWritable := 'False'} : Word;
   //    InterfaceInformation : "LPNDR_typeInterfaceInformation";
   //    PortInformation : Array[1..52] of "LPNDR_typePortInformation";
   //    PortLinkState : Array[1..52] of "LPNDR_typePortLinkState";
   //    PortStatistic : Array[1..52] of "LPNDR_typePortStatistic";
   //    diagnostics { ExternalWritable := 'False'} : "typeDiagnostics";
   // END_VAR
   // VAR
   //    statExecuteOld { ExternalAccessible := 'False'; ExternalVisible := 'False'; ExternalWritable := 'False'} : Bool;
   //    statDone { ExternalAccessible := 'False'; ExternalVisible := 'False'; ExternalWritable := 'False'} : Bool;
   //    statBusy { ExternalAccessible := 'False'; ExternalVisible := 'False'; ExternalWritable := 'False'} : Bool;
   //    statError { ExternalAccessible := 'False'; ExternalVisible := 'False'; ExternalWritable := 'False'} : Bool;
   //    statStatus { ExternalAccessible := 'False'; ExternalVisible := 'False'; ExternalWritable := 'False'} : Word;
   //    statSubfunctionStatus { ExternalAccessible := 'False'; ExternalVisible := 'False'; ExternalWritable := 'False'} : Word;
   //    statFBErrorState { ExternalAccessible := 'False'; ExternalVisible := 'False'; ExternalWritable := 'False'} : DInt;
   //    statFBState { ExternalAccessible := 'False'; ExternalVisible := 'False'; ExternalWritable := 'False'} : DInt;
   //    statEmptyDiagnostics { ExternalAccessible := 'False'; ExternalVisible := 'False'; ExternalWritable := 'False'} : "typeDiagnostics";
   //    InstReadRecord { S7_SetPoint := 'True'} : RDREC;
   //    statReadRecordLength : UInt;
   //    statReadRecordRequest : Bool;
   //    statPDInterfaceMrpDataReal : UInt;
   //    statPDPortMrpDataReal : UInt;
   //    statPDInterfaceDataReal : UInt;
   //    statPDPortDataReal : UInt;
   //    statPDPortStatistic : UInt;
   //    statUnknown : UInt;
   //    statInterfaceInfoReset : "LPNDR_typeInterfaceInformation";
   //    statPortInfoReset { S7_SetPoint := 'True'} : "LPNDR_typePortInformation";
   //    statPortLinkStateReset { S7_SetPoint := 'True'} : "LPNDR_typePortLinkState";
   //    statPortStatisticReset { S7_SetPoint := 'True'} : "LPNDR_typePortStatistic";
   //    statReadRecord { S7_SetPoint := 'True'} : Array[0..4175] of Byte;
   // END_VAR
BEGIN
END_DATA_BLOCK

DATA_BLOCK "Main_Safety_RTG1_DB"   // DB501, F_DB
NAME : FUSI
VERSION : 0.1
// stored: AutoNumber false, DBAccessibleFromOPCUA true, DBAccessibleFromWebserver true, InstanceOfName Main_Safety_RTG1, InstanceOfType FB
"Main_Safety_RTG1"
BEGIN
END_DATA_BLOCK

DATA_BLOCK "MbBMS1"   // DB26
// stored: AutoNumber false, DBAccessibleFromOPCUA true, DBAccessibleFromWebserver true, InstanceOfName MB_CLIENT, OfSystemLibElement MB_CLIENT, OfSystemLibVersion 5.2
"MB_CLIENT"
   // VAR_INPUT
   //    REQ : Bool;
   //    DISCONNECT : Bool;
   //    MB_MODE : USInt;
   //    MB_DATA_ADDR : UDInt;
   //    MB_DATA_LEN : UInt;
   // END_VAR
   // VAR_OUTPUT
   //    DONE : Bool;
   //    BUSY : Bool;
   //    ERROR : Bool;
   //    STATUS { ExternalVisible := 'False'} : Word;
   // END_VAR
   // VAR_IN_OUT
   //    MB_DATA_PTR : Variant;
   //    CONNECT : Variant;
   // END_VAR
   // VAR
   //    TCON { S7_SetPoint := 'True'} : TCON;
   //    TDISCON { S7_SetPoint := 'True'} : TDISCON;
   //    TSEND { S7_SetPoint := 'True'} : TSEND;
   //    TRECEIVE { S7_SetPoint := 'True'} : TRCV;
   //    TRESET { S7_SetPoint := 'True'} : T_RESET;
   //    TDIAG { S7_SetPoint := 'True'} : T_DIAG;
   //    TDIAG_Status { S7_SetPoint := 'True'} : TDiag_Status;
   //    Blocked_Proc_Timeout : Real;
   //    Rcv_Timeout : Real;
   //    MB_Unit_ID : Byte;
   //    MB_Transaction_ID : Word;
   //    MB_State { ExternalWritable := 'False'} : Word;
   //    SAVED_MB_DATA_ADDR : UDInt;
   //    SAVED_DATA_LEN : UInt;
   //    SAVED_MB_MODE : USInt;
   //    Connection_ID : Word;
   //    Retries : Word;
   //    TEMP_DATA { ExternalWritable := 'False'} : Array[1..263] of Byte;
   //    rcv_timer { ExternalAccessible := 'False'; ExternalVisible := 'False'; ExternalWritable := 'False'; S7_SetPoint := 'True'} : TON_TIME;
   //    wd_timer { ExternalAccessible := 'False'; ExternalVisible := 'False'; ExternalWritable := 'False'; S7_SetPoint := 'True'} : TON_TIME;
   //    Connected : Bool;
   //    Active { ExternalWritable := 'False'} : Bool;
   //    BytesReceived : UDInt;
   // END_VAR
BEGIN
END_DATA_BLOCK

DATA_BLOCK "MbBMS10"   // DB24
// stored: AutoNumber false, DBAccessibleFromOPCUA true, DBAccessibleFromWebserver true, InstanceOfName MB_CLIENT, OfSystemLibElement MB_CLIENT, OfSystemLibVersion 5.2
"MB_CLIENT"
   // VAR_INPUT
   //    REQ : Bool;
   //    DISCONNECT : Bool;
   //    MB_MODE : USInt;
   //    MB_DATA_ADDR : UDInt;
   //    MB_DATA_LEN : UInt;
   // END_VAR
   // VAR_OUTPUT
   //    DONE : Bool;
   //    BUSY : Bool;
   //    ERROR : Bool;
   //    STATUS { ExternalVisible := 'False'} : Word;
   // END_VAR
   // VAR_IN_OUT
   //    MB_DATA_PTR : Variant;
   //    CONNECT : Variant;
   // END_VAR
   // VAR
   //    TCON { S7_SetPoint := 'True'} : TCON;
   //    TDISCON { S7_SetPoint := 'True'} : TDISCON;
   //    TSEND { S7_SetPoint := 'True'} : TSEND;
   //    TRECEIVE { S7_SetPoint := 'True'} : TRCV;
   //    TRESET { S7_SetPoint := 'True'} : T_RESET;
   //    TDIAG { S7_SetPoint := 'True'} : T_DIAG;
   //    TDIAG_Status { S7_SetPoint := 'True'} : TDiag_Status;
   //    Blocked_Proc_Timeout : Real;
   //    Rcv_Timeout : Real;
   //    MB_Unit_ID : Byte;
   //    MB_Transaction_ID : Word;
   //    MB_State { ExternalWritable := 'False'} : Word;
   //    SAVED_MB_DATA_ADDR : UDInt;
   //    SAVED_DATA_LEN : UInt;
   //    SAVED_MB_MODE : USInt;
   //    Connection_ID : Word;
   //    Retries : Word;
   //    TEMP_DATA { ExternalWritable := 'False'} : Array[1..263] of Byte;
   //    rcv_timer { ExternalAccessible := 'False'; ExternalVisible := 'False'; ExternalWritable := 'False'; S7_SetPoint := 'True'} : TON_TIME;
   //    wd_timer { ExternalAccessible := 'False'; ExternalVisible := 'False'; ExternalWritable := 'False'; S7_SetPoint := 'True'} : TON_TIME;
   //    Connected : Bool;
   //    Active { ExternalWritable := 'False'} : Bool;
   //    BytesReceived : UDInt;
   // END_VAR
BEGIN
END_DATA_BLOCK

DATA_BLOCK "MbBMS11"   // DB25
// stored: AutoNumber false, DBAccessibleFromOPCUA true, DBAccessibleFromWebserver true, InstanceOfName MB_CLIENT, OfSystemLibElement MB_CLIENT, OfSystemLibVersion 5.2
"MB_CLIENT"
   // VAR_INPUT
   //    REQ : Bool;
   //    DISCONNECT : Bool;
   //    MB_MODE : USInt;
   //    MB_DATA_ADDR : UDInt;
   //    MB_DATA_LEN : UInt;
   // END_VAR
   // VAR_OUTPUT
   //    DONE : Bool;
   //    BUSY : Bool;
   //    ERROR : Bool;
   //    STATUS { ExternalVisible := 'False'} : Word;
   // END_VAR
   // VAR_IN_OUT
   //    MB_DATA_PTR : Variant;
   //    CONNECT : Variant;
   // END_VAR
   // VAR
   //    TCON { S7_SetPoint := 'True'} : TCON;
   //    TDISCON { S7_SetPoint := 'True'} : TDISCON;
   //    TSEND { S7_SetPoint := 'True'} : TSEND;
   //    TRECEIVE { S7_SetPoint := 'True'} : TRCV;
   //    TRESET { S7_SetPoint := 'True'} : T_RESET;
   //    TDIAG { S7_SetPoint := 'True'} : T_DIAG;
   //    TDIAG_Status { S7_SetPoint := 'True'} : TDiag_Status;
   //    Blocked_Proc_Timeout : Real;
   //    Rcv_Timeout : Real;
   //    MB_Unit_ID : Byte;
   //    MB_Transaction_ID : Word;
   //    MB_State { ExternalWritable := 'False'} : Word;
   //    SAVED_MB_DATA_ADDR : UDInt;
   //    SAVED_DATA_LEN : UInt;
   //    SAVED_MB_MODE : USInt;
   //    Connection_ID : Word;
   //    Retries : Word;
   //    TEMP_DATA { ExternalWritable := 'False'} : Array[1..263] of Byte;
   //    rcv_timer { ExternalAccessible := 'False'; ExternalVisible := 'False'; ExternalWritable := 'False'; S7_SetPoint := 'True'} : TON_TIME;
   //    wd_timer { ExternalAccessible := 'False'; ExternalVisible := 'False'; ExternalWritable := 'False'; S7_SetPoint := 'True'} : TON_TIME;
   //    Connected : Bool;
   //    Active { ExternalWritable := 'False'} : Bool;
   //    BytesReceived : UDInt;
   // END_VAR
BEGIN
END_DATA_BLOCK

DATA_BLOCK "MbBMS2"   // DB29
// stored: AutoNumber false, DBAccessibleFromOPCUA true, DBAccessibleFromWebserver true, InstanceOfName MB_CLIENT, OfSystemLibElement MB_CLIENT, OfSystemLibVersion 5.2
"MB_CLIENT"
   // VAR_INPUT
   //    REQ : Bool;
   //    DISCONNECT : Bool;
   //    MB_MODE : USInt;
   //    MB_DATA_ADDR : UDInt;
   //    MB_DATA_LEN : UInt;
   // END_VAR
   // VAR_OUTPUT
   //    DONE : Bool;
   //    BUSY : Bool;
   //    ERROR : Bool;
   //    STATUS { ExternalVisible := 'False'} : Word;
   // END_VAR
   // VAR_IN_OUT
   //    MB_DATA_PTR : Variant;
   //    CONNECT : Variant;
   // END_VAR
   // VAR
   //    TCON { S7_SetPoint := 'True'} : TCON;
   //    TDISCON { S7_SetPoint := 'True'} : TDISCON;
   //    TSEND { S7_SetPoint := 'True'} : TSEND;
   //    TRECEIVE { S7_SetPoint := 'True'} : TRCV;
   //    TRESET { S7_SetPoint := 'True'} : T_RESET;
   //    TDIAG { S7_SetPoint := 'True'} : T_DIAG;
   //    TDIAG_Status { S7_SetPoint := 'True'} : TDiag_Status;
   //    Blocked_Proc_Timeout : Real;
   //    Rcv_Timeout : Real;
   //    MB_Unit_ID : Byte;
   //    MB_Transaction_ID : Word;
   //    MB_State { ExternalWritable := 'False'} : Word;
   //    SAVED_MB_DATA_ADDR : UDInt;
   //    SAVED_DATA_LEN : UInt;
   //    SAVED_MB_MODE : USInt;
   //    Connection_ID : Word;
   //    Retries : Word;
   //    TEMP_DATA { ExternalWritable := 'False'} : Array[1..263] of Byte;
   //    rcv_timer { ExternalAccessible := 'False'; ExternalVisible := 'False'; ExternalWritable := 'False'; S7_SetPoint := 'True'} : TON_TIME;
   //    wd_timer { ExternalAccessible := 'False'; ExternalVisible := 'False'; ExternalWritable := 'False'; S7_SetPoint := 'True'} : TON_TIME;
   //    Connected : Bool;
   //    Active { ExternalWritable := 'False'} : Bool;
   //    BytesReceived : UDInt;
   // END_VAR
BEGIN
END_DATA_BLOCK

DATA_BLOCK "MbBMS20"   // DB27
// stored: AutoNumber false, DBAccessibleFromOPCUA true, DBAccessibleFromWebserver true, InstanceOfName MB_CLIENT, OfSystemLibElement MB_CLIENT, OfSystemLibVersion 5.2
"MB_CLIENT"
   // VAR_INPUT
   //    REQ : Bool;
   //    DISCONNECT : Bool;
   //    MB_MODE : USInt;
   //    MB_DATA_ADDR : UDInt;
   //    MB_DATA_LEN : UInt;
   // END_VAR
   // VAR_OUTPUT
   //    DONE : Bool;
   //    BUSY : Bool;
   //    ERROR : Bool;
   //    STATUS { ExternalVisible := 'False'} : Word;
   // END_VAR
   // VAR_IN_OUT
   //    MB_DATA_PTR : Variant;
   //    CONNECT : Variant;
   // END_VAR
   // VAR
   //    TCON { S7_SetPoint := 'True'} : TCON;
   //    TDISCON { S7_SetPoint := 'True'} : TDISCON;
   //    TSEND { S7_SetPoint := 'True'} : TSEND;
   //    TRECEIVE { S7_SetPoint := 'True'} : TRCV;
   //    TRESET { S7_SetPoint := 'True'} : T_RESET;
   //    TDIAG { S7_SetPoint := 'True'} : T_DIAG;
   //    TDIAG_Status { S7_SetPoint := 'True'} : TDiag_Status;
   //    Blocked_Proc_Timeout : Real;
   //    Rcv_Timeout : Real;
   //    MB_Unit_ID : Byte;
   //    MB_Transaction_ID : Word;
   //    MB_State { ExternalWritable := 'False'} : Word;
   //    SAVED_MB_DATA_ADDR : UDInt;
   //    SAVED_DATA_LEN : UInt;
   //    SAVED_MB_MODE : USInt;
   //    Connection_ID : Word;
   //    Retries : Word;
   //    TEMP_DATA { ExternalWritable := 'False'} : Array[1..263] of Byte;
   //    rcv_timer { ExternalAccessible := 'False'; ExternalVisible := 'False'; ExternalWritable := 'False'; S7_SetPoint := 'True'} : TON_TIME;
   //    wd_timer { ExternalAccessible := 'False'; ExternalVisible := 'False'; ExternalWritable := 'False'; S7_SetPoint := 'True'} : TON_TIME;
   //    Connected : Bool;
   //    Active { ExternalWritable := 'False'} : Bool;
   //    BytesReceived : UDInt;
   // END_VAR
BEGIN
END_DATA_BLOCK

DATA_BLOCK "MbBMS21"   // DB28
// stored: AutoNumber false, DBAccessibleFromOPCUA true, DBAccessibleFromWebserver true, InstanceOfName MB_CLIENT, OfSystemLibElement MB_CLIENT, OfSystemLibVersion 5.2
"MB_CLIENT"
   // VAR_INPUT
   //    REQ : Bool;
   //    DISCONNECT : Bool;
   //    MB_MODE : USInt;
   //    MB_DATA_ADDR : UDInt;
   //    MB_DATA_LEN : UInt;
   // END_VAR
   // VAR_OUTPUT
   //    DONE : Bool;
   //    BUSY : Bool;
   //    ERROR : Bool;
   //    STATUS { ExternalVisible := 'False'} : Word;
   // END_VAR
   // VAR_IN_OUT
   //    MB_DATA_PTR : Variant;
   //    CONNECT : Variant;
   // END_VAR
   // VAR
   //    TCON { S7_SetPoint := 'True'} : TCON;
   //    TDISCON { S7_SetPoint := 'True'} : TDISCON;
   //    TSEND { S7_SetPoint := 'True'} : TSEND;
   //    TRECEIVE { S7_SetPoint := 'True'} : TRCV;
   //    TRESET { S7_SetPoint := 'True'} : T_RESET;
   //    TDIAG { S7_SetPoint := 'True'} : T_DIAG;
   //    TDIAG_Status { S7_SetPoint := 'True'} : TDiag_Status;
   //    Blocked_Proc_Timeout : Real;
   //    Rcv_Timeout : Real;
   //    MB_Unit_ID : Byte;
   //    MB_Transaction_ID : Word;
   //    MB_State { ExternalWritable := 'False'} : Word;
   //    SAVED_MB_DATA_ADDR : UDInt;
   //    SAVED_DATA_LEN : UInt;
   //    SAVED_MB_MODE : USInt;
   //    Connection_ID : Word;
   //    Retries : Word;
   //    TEMP_DATA { ExternalWritable := 'False'} : Array[1..263] of Byte;
   //    rcv_timer { ExternalAccessible := 'False'; ExternalVisible := 'False'; ExternalWritable := 'False'; S7_SetPoint := 'True'} : TON_TIME;
   //    wd_timer { ExternalAccessible := 'False'; ExternalVisible := 'False'; ExternalWritable := 'False'; S7_SetPoint := 'True'} : TON_TIME;
   //    Connected : Bool;
   //    Active { ExternalWritable := 'False'} : Bool;
   //    BytesReceived : UDInt;
   // END_VAR
BEGIN
END_DATA_BLOCK

DATA_BLOCK "MbMVSKID"   // DB46
// stored: AutoNumber false, DBAccessibleFromOPCUA true, DBAccessibleFromWebserver true, InstanceOfName MB_CLIENT, OfSystemLibElement MB_CLIENT, OfSystemLibVersion 5.2
"MB_CLIENT"
   // VAR_INPUT
   //    REQ : Bool;
   //    DISCONNECT : Bool;
   //    MB_MODE : USInt;
   //    MB_DATA_ADDR : UDInt;
   //    MB_DATA_LEN : UInt;
   // END_VAR
   // VAR_OUTPUT
   //    DONE : Bool;
   //    BUSY : Bool;
   //    ERROR : Bool;
   //    STATUS { ExternalVisible := 'False'} : Word;
   // END_VAR
   // VAR_IN_OUT
   //    MB_DATA_PTR : Variant;
   //    CONNECT : Variant;
   // END_VAR
   // VAR
   //    TCON { S7_SetPoint := 'True'} : TCON;
   //    TDISCON { S7_SetPoint := 'True'} : TDISCON;
   //    TSEND { S7_SetPoint := 'True'} : TSEND;
   //    TRECEIVE { S7_SetPoint := 'True'} : TRCV;
   //    TRESET { S7_SetPoint := 'True'} : T_RESET;
   //    TDIAG { S7_SetPoint := 'True'} : T_DIAG;
   //    TDIAG_Status { S7_SetPoint := 'True'} : TDiag_Status;
   //    Blocked_Proc_Timeout : Real;
   //    Rcv_Timeout : Real;
   //    MB_Unit_ID : Byte;
   //    MB_Transaction_ID : Word;
   //    MB_State { ExternalWritable := 'False'} : Word;
   //    SAVED_MB_DATA_ADDR : UDInt;
   //    SAVED_DATA_LEN : UInt;
   //    SAVED_MB_MODE : USInt;
   //    Connection_ID : Word;
   //    Retries : Word;
   //    TEMP_DATA { ExternalWritable := 'False'} : Array[1..263] of Byte;
   //    rcv_timer { ExternalAccessible := 'False'; ExternalVisible := 'False'; ExternalWritable := 'False'; S7_SetPoint := 'True'} : TON_TIME;
   //    wd_timer { ExternalAccessible := 'False'; ExternalVisible := 'False'; ExternalWritable := 'False'; S7_SetPoint := 'True'} : TON_TIME;
   //    Connected : Bool;
   //    Active { ExternalWritable := 'False'} : Bool;
   //    BytesReceived : UDInt;
   // END_VAR
BEGIN
END_DATA_BLOCK

DATA_BLOCK "MbMVSKID_1"   // DB7
// stored: AutoNumber true, DBAccessibleFromOPCUA true, DBAccessibleFromWebserver true, InstanceOfName MB_CLIENT, OfSystemLibElement MB_CLIENT, OfSystemLibVersion 5.2
"MB_CLIENT"
   // VAR_INPUT
   //    REQ : Bool;
   //    DISCONNECT : Bool;
   //    MB_MODE : USInt;
   //    MB_DATA_ADDR : UDInt;
   //    MB_DATA_LEN : UInt;
   // END_VAR
   // VAR_OUTPUT
   //    DONE : Bool;
   //    BUSY : Bool;
   //    ERROR : Bool;
   //    STATUS { ExternalVisible := 'False'} : Word;
   // END_VAR
   // VAR_IN_OUT
   //    MB_DATA_PTR : Variant;
   //    CONNECT : Variant;
   // END_VAR
   // VAR
   //    TCON { S7_SetPoint := 'True'} : TCON;
   //    TDISCON { S7_SetPoint := 'True'} : TDISCON;
   //    TSEND { S7_SetPoint := 'True'} : TSEND;
   //    TRECEIVE { S7_SetPoint := 'True'} : TRCV;
   //    TRESET { S7_SetPoint := 'True'} : T_RESET;
   //    TDIAG { S7_SetPoint := 'True'} : T_DIAG;
   //    TDIAG_Status { S7_SetPoint := 'True'} : TDiag_Status;
   //    Blocked_Proc_Timeout : Real;
   //    Rcv_Timeout : Real;
   //    MB_Unit_ID : Byte;
   //    MB_Transaction_ID : Word;
   //    MB_State { ExternalWritable := 'False'} : Word;
   //    SAVED_MB_DATA_ADDR : UDInt;
   //    SAVED_DATA_LEN : UInt;
   //    SAVED_MB_MODE : USInt;
   //    Connection_ID : Word;
   //    Retries : Word;
   //    TEMP_DATA { ExternalWritable := 'False'} : Array[1..263] of Byte;
   //    rcv_timer { ExternalAccessible := 'False'; ExternalVisible := 'False'; ExternalWritable := 'False'; S7_SetPoint := 'True'} : TON_TIME;
   //    wd_timer { ExternalAccessible := 'False'; ExternalVisible := 'False'; ExternalWritable := 'False'; S7_SetPoint := 'True'} : TON_TIME;
   //    Connected : Bool;
   //    Active { ExternalWritable := 'False'} : Bool;
   //    BytesReceived : UDInt;
   // END_VAR
BEGIN
END_DATA_BLOCK

DATA_BLOCK "MbMVSKID_2"   // DB8
// stored: AutoNumber true, DBAccessibleFromOPCUA true, DBAccessibleFromWebserver true, InstanceOfName MB_CLIENT, OfSystemLibElement MB_CLIENT, OfSystemLibVersion 5.2
"MB_CLIENT"
   // VAR_INPUT
   //    REQ : Bool;
   //    DISCONNECT : Bool;
   //    MB_MODE : USInt;
   //    MB_DATA_ADDR : UDInt;
   //    MB_DATA_LEN : UInt;
   // END_VAR
   // VAR_OUTPUT
   //    DONE : Bool;
   //    BUSY : Bool;
   //    ERROR : Bool;
   //    STATUS { ExternalVisible := 'False'} : Word;
   // END_VAR
   // VAR_IN_OUT
   //    MB_DATA_PTR : Variant;
   //    CONNECT : Variant;
   // END_VAR
   // VAR
   //    TCON { S7_SetPoint := 'True'} : TCON;
   //    TDISCON { S7_SetPoint := 'True'} : TDISCON;
   //    TSEND { S7_SetPoint := 'True'} : TSEND;
   //    TRECEIVE { S7_SetPoint := 'True'} : TRCV;
   //    TRESET { S7_SetPoint := 'True'} : T_RESET;
   //    TDIAG { S7_SetPoint := 'True'} : T_DIAG;
   //    TDIAG_Status { S7_SetPoint := 'True'} : TDiag_Status;
   //    Blocked_Proc_Timeout : Real;
   //    Rcv_Timeout : Real;
   //    MB_Unit_ID : Byte;
   //    MB_Transaction_ID : Word;
   //    MB_State { ExternalWritable := 'False'} : Word;
   //    SAVED_MB_DATA_ADDR : UDInt;
   //    SAVED_DATA_LEN : UInt;
   //    SAVED_MB_MODE : USInt;
   //    Connection_ID : Word;
   //    Retries : Word;
   //    TEMP_DATA { ExternalWritable := 'False'} : Array[1..263] of Byte;
   //    rcv_timer { ExternalAccessible := 'False'; ExternalVisible := 'False'; ExternalWritable := 'False'; S7_SetPoint := 'True'} : TON_TIME;
   //    wd_timer { ExternalAccessible := 'False'; ExternalVisible := 'False'; ExternalWritable := 'False'; S7_SetPoint := 'True'} : TON_TIME;
   //    Connected : Bool;
   //    Active { ExternalWritable := 'False'} : Bool;
   //    BytesReceived : UDInt;
   // END_VAR
BEGIN
END_DATA_BLOCK

DATA_BLOCK "MbPCS1"   // DB45
// stored: AutoNumber false, DBAccessibleFromOPCUA true, DBAccessibleFromWebserver true, InstanceOfName MB_CLIENT, OfSystemLibElement MB_CLIENT, OfSystemLibVersion 5.2
"MB_CLIENT"
   // VAR_INPUT
   //    REQ : Bool;
   //    DISCONNECT : Bool;
   //    MB_MODE : USInt;
   //    MB_DATA_ADDR : UDInt;
   //    MB_DATA_LEN : UInt;
   // END_VAR
   // VAR_OUTPUT
   //    DONE : Bool;
   //    BUSY : Bool;
   //    ERROR : Bool;
   //    STATUS { ExternalVisible := 'False'} : Word;
   // END_VAR
   // VAR_IN_OUT
   //    MB_DATA_PTR : Variant;
   //    CONNECT : Variant;
   // END_VAR
   // VAR
   //    TCON { S7_SetPoint := 'True'} : TCON;
   //    TDISCON { S7_SetPoint := 'True'} : TDISCON;
   //    TSEND { S7_SetPoint := 'True'} : TSEND;
   //    TRECEIVE { S7_SetPoint := 'True'} : TRCV;
   //    TRESET { S7_SetPoint := 'True'} : T_RESET;
   //    TDIAG { S7_SetPoint := 'True'} : T_DIAG;
   //    TDIAG_Status { S7_SetPoint := 'True'} : TDiag_Status;
   //    Blocked_Proc_Timeout : Real;
   //    Rcv_Timeout : Real;
   //    MB_Unit_ID : Byte;
   //    MB_Transaction_ID : Word;
   //    MB_State { ExternalWritable := 'False'} : Word;
   //    SAVED_MB_DATA_ADDR : UDInt;
   //    SAVED_DATA_LEN : UInt;
   //    SAVED_MB_MODE : USInt;
   //    Connection_ID : Word;
   //    Retries : Word;
   //    TEMP_DATA { ExternalWritable := 'False'} : Array[1..263] of Byte;
   //    rcv_timer { ExternalAccessible := 'False'; ExternalVisible := 'False'; ExternalWritable := 'False'; S7_SetPoint := 'True'} : TON_TIME;
   //    wd_timer { ExternalAccessible := 'False'; ExternalVisible := 'False'; ExternalWritable := 'False'; S7_SetPoint := 'True'} : TON_TIME;
   //    Connected : Bool;
   //    Active { ExternalWritable := 'False'} : Bool;
   //    BytesReceived : UDInt;
   // END_VAR
BEGIN
END_DATA_BLOCK

DATA_BLOCK "MbPCS10"   // DB44
// stored: AutoNumber false, DBAccessibleFromOPCUA true, DBAccessibleFromWebserver true, InstanceOfName MB_CLIENT, OfSystemLibElement MB_CLIENT, OfSystemLibVersion 5.2
"MB_CLIENT"
   // VAR_INPUT
   //    REQ : Bool;
   //    DISCONNECT : Bool;
   //    MB_MODE : USInt;
   //    MB_DATA_ADDR : UDInt;
   //    MB_DATA_LEN : UInt;
   // END_VAR
   // VAR_OUTPUT
   //    DONE : Bool;
   //    BUSY : Bool;
   //    ERROR : Bool;
   //    STATUS { ExternalVisible := 'False'} : Word;
   // END_VAR
   // VAR_IN_OUT
   //    MB_DATA_PTR : Variant;
   //    CONNECT : Variant;
   // END_VAR
   // VAR
   //    TCON { S7_SetPoint := 'True'} : TCON;
   //    TDISCON { S7_SetPoint := 'True'} : TDISCON;
   //    TSEND { S7_SetPoint := 'True'} : TSEND;
   //    TRECEIVE { S7_SetPoint := 'True'} : TRCV;
   //    TRESET { S7_SetPoint := 'True'} : T_RESET;
   //    TDIAG { S7_SetPoint := 'True'} : T_DIAG;
   //    TDIAG_Status { S7_SetPoint := 'True'} : TDiag_Status;
   //    Blocked_Proc_Timeout : Real;
   //    Rcv_Timeout : Real;
   //    MB_Unit_ID : Byte;
   //    MB_Transaction_ID : Word;
   //    MB_State { ExternalWritable := 'False'} : Word;
   //    SAVED_MB_DATA_ADDR : UDInt;
   //    SAVED_DATA_LEN : UInt;
   //    SAVED_MB_MODE : USInt;
   //    Connection_ID : Word;
   //    Retries : Word;
   //    TEMP_DATA { ExternalWritable := 'False'} : Array[1..263] of Byte;
   //    rcv_timer { ExternalAccessible := 'False'; ExternalVisible := 'False'; ExternalWritable := 'False'; S7_SetPoint := 'True'} : TON_TIME;
   //    wd_timer { ExternalAccessible := 'False'; ExternalVisible := 'False'; ExternalWritable := 'False'; S7_SetPoint := 'True'} : TON_TIME;
   //    Connected : Bool;
   //    Active { ExternalWritable := 'False'} : Bool;
   //    BytesReceived : UDInt;
   // END_VAR
BEGIN
END_DATA_BLOCK

DATA_BLOCK "MbPCS1_W"   // DB43
// stored: AutoNumber false, DBAccessibleFromOPCUA true, DBAccessibleFromWebserver true, InstanceOfName MB_CLIENT, OfSystemLibElement MB_CLIENT, OfSystemLibVersion 5.2
"MB_CLIENT"
   // VAR_INPUT
   //    REQ : Bool;
   //    DISCONNECT : Bool;
   //    MB_MODE : USInt;
   //    MB_DATA_ADDR : UDInt;
   //    MB_DATA_LEN : UInt;
   // END_VAR
   // VAR_OUTPUT
   //    DONE : Bool;
   //    BUSY : Bool;
   //    ERROR : Bool;
   //    STATUS { ExternalVisible := 'False'} : Word;
   // END_VAR
   // VAR_IN_OUT
   //    MB_DATA_PTR : Variant;
   //    CONNECT : Variant;
   // END_VAR
   // VAR
   //    TCON { S7_SetPoint := 'True'} : TCON;
   //    TDISCON { S7_SetPoint := 'True'} : TDISCON;
   //    TSEND { S7_SetPoint := 'True'} : TSEND;
   //    TRECEIVE { S7_SetPoint := 'True'} : TRCV;
   //    TRESET { S7_SetPoint := 'True'} : T_RESET;
   //    TDIAG { S7_SetPoint := 'True'} : T_DIAG;
   //    TDIAG_Status { S7_SetPoint := 'True'} : TDiag_Status;
   //    Blocked_Proc_Timeout : Real;
   //    Rcv_Timeout : Real;
   //    MB_Unit_ID : Byte;
   //    MB_Transaction_ID : Word;
   //    MB_State { ExternalWritable := 'False'} : Word;
   //    SAVED_MB_DATA_ADDR : UDInt;
   //    SAVED_DATA_LEN : UInt;
   //    SAVED_MB_MODE : USInt;
   //    Connection_ID : Word;
   //    Retries : Word;
   //    TEMP_DATA { ExternalWritable := 'False'} : Array[1..263] of Byte;
   //    rcv_timer { ExternalAccessible := 'False'; ExternalVisible := 'False'; ExternalWritable := 'False'; S7_SetPoint := 'True'} : TON_TIME;
   //    wd_timer { ExternalAccessible := 'False'; ExternalVisible := 'False'; ExternalWritable := 'False'; S7_SetPoint := 'True'} : TON_TIME;
   //    Connected : Bool;
   //    Active { ExternalWritable := 'False'} : Bool;
   //    BytesReceived : UDInt;
   // END_VAR
BEGIN
END_DATA_BLOCK

DATA_BLOCK "MbPCS_1-R_fast"   // DB44
// stored: AutoNumber false, DBAccessibleFromOPCUA true, DBAccessibleFromWebserver true, InstanceOfName MB_CLIENT, OfSystemLibElement MB_CLIENT, OfSystemLibVersion 5.2
"MB_CLIENT"
   // VAR_INPUT
   //    REQ : Bool;
   //    DISCONNECT : Bool;
   //    MB_MODE : USInt;
   //    MB_DATA_ADDR : UDInt;
   //    MB_DATA_LEN : UInt;
   // END_VAR
   // VAR_OUTPUT
   //    DONE : Bool;
   //    BUSY : Bool;
   //    ERROR : Bool;
   //    STATUS { ExternalVisible := 'False'} : Word;
   // END_VAR
   // VAR_IN_OUT
   //    MB_DATA_PTR : Variant;
   //    CONNECT : Variant;
   // END_VAR
   // VAR
   //    TCON { S7_SetPoint := 'True'} : TCON;
   //    TDISCON { S7_SetPoint := 'True'} : TDISCON;
   //    TSEND { S7_SetPoint := 'True'} : TSEND;
   //    TRECEIVE { S7_SetPoint := 'True'} : TRCV;
   //    TRESET { S7_SetPoint := 'True'} : T_RESET;
   //    TDIAG { S7_SetPoint := 'True'} : T_DIAG;
   //    TDIAG_Status { S7_SetPoint := 'True'} : TDiag_Status;
   //    Blocked_Proc_Timeout : Real;
   //    Rcv_Timeout : Real;
   //    MB_Unit_ID : Byte;
   //    MB_Transaction_ID : Word;
   //    MB_State { ExternalWritable := 'False'} : Word;
   //    SAVED_MB_DATA_ADDR : UDInt;
   //    SAVED_DATA_LEN : UInt;
   //    SAVED_MB_MODE : USInt;
   //    Connection_ID : Word;
   //    Retries : Word;
   //    TEMP_DATA { ExternalWritable := 'False'} : Array[1..263] of Byte;
   //    rcv_timer { ExternalAccessible := 'False'; ExternalVisible := 'False'; ExternalWritable := 'False'; S7_SetPoint := 'True'} : TON_TIME;
   //    wd_timer { ExternalAccessible := 'False'; ExternalVisible := 'False'; ExternalWritable := 'False'; S7_SetPoint := 'True'} : TON_TIME;
   //    Connected : Bool;
   //    Active { ExternalWritable := 'False'} : Bool;
   //    BytesReceived : UDInt;
   // END_VAR
BEGIN
END_DATA_BLOCK

DATA_BLOCK "MbPCS_1-R_slow"   // DB45
// stored: AutoNumber false, DBAccessibleFromOPCUA true, DBAccessibleFromWebserver true, InstanceOfName MB_CLIENT, OfSystemLibElement MB_CLIENT, OfSystemLibVersion 5.2
"MB_CLIENT"
   // VAR_INPUT
   //    REQ : Bool;
   //    DISCONNECT : Bool;
   //    MB_MODE : USInt;
   //    MB_DATA_ADDR : UDInt;
   //    MB_DATA_LEN : UInt;
   // END_VAR
   // VAR_OUTPUT
   //    DONE : Bool;
   //    BUSY : Bool;
   //    ERROR : Bool;
   //    STATUS { ExternalVisible := 'False'} : Word;
   // END_VAR
   // VAR_IN_OUT
   //    MB_DATA_PTR : Variant;
   //    CONNECT : Variant;
   // END_VAR
   // VAR
   //    TCON { S7_SetPoint := 'True'} : TCON;
   //    TDISCON { S7_SetPoint := 'True'} : TDISCON;
   //    TSEND { S7_SetPoint := 'True'} : TSEND;
   //    TRECEIVE { S7_SetPoint := 'True'} : TRCV;
   //    TRESET { S7_SetPoint := 'True'} : T_RESET;
   //    TDIAG { S7_SetPoint := 'True'} : T_DIAG;
   //    TDIAG_Status { S7_SetPoint := 'True'} : TDiag_Status;
   //    Blocked_Proc_Timeout : Real;
   //    Rcv_Timeout : Real;
   //    MB_Unit_ID : Byte;
   //    MB_Transaction_ID : Word;
   //    MB_State { ExternalWritable := 'False'} : Word;
   //    SAVED_MB_DATA_ADDR : UDInt;
   //    SAVED_DATA_LEN : UInt;
   //    SAVED_MB_MODE : USInt;
   //    Connection_ID : Word;
   //    Retries : Word;
   //    TEMP_DATA { ExternalWritable := 'False'} : Array[1..263] of Byte;
   //    rcv_timer { ExternalAccessible := 'False'; ExternalVisible := 'False'; ExternalWritable := 'False'; S7_SetPoint := 'True'} : TON_TIME;
   //    wd_timer { ExternalAccessible := 'False'; ExternalVisible := 'False'; ExternalWritable := 'False'; S7_SetPoint := 'True'} : TON_TIME;
   //    Connected : Bool;
   //    Active { ExternalWritable := 'False'} : Bool;
   //    BytesReceived : UDInt;
   // END_VAR
BEGIN
END_DATA_BLOCK

DATA_BLOCK "MbPCS_1-W_fast"   // DB5
// stored: AutoNumber true, DBAccessibleFromOPCUA true, DBAccessibleFromWebserver true, InstanceOfName MB_CLIENT, OfSystemLibElement MB_CLIENT, OfSystemLibVersion 5.2
"MB_CLIENT"
   // VAR_INPUT
   //    REQ : Bool;
   //    DISCONNECT : Bool;
   //    MB_MODE : USInt;
   //    MB_DATA_ADDR : UDInt;
   //    MB_DATA_LEN : UInt;
   // END_VAR
   // VAR_OUTPUT
   //    DONE : Bool;
   //    BUSY : Bool;
   //    ERROR : Bool;
   //    STATUS { ExternalVisible := 'False'} : Word;
   // END_VAR
   // VAR_IN_OUT
   //    MB_DATA_PTR : Variant;
   //    CONNECT : Variant;
   // END_VAR
   // VAR
   //    TCON { S7_SetPoint := 'True'} : TCON;
   //    TDISCON { S7_SetPoint := 'True'} : TDISCON;
   //    TSEND { S7_SetPoint := 'True'} : TSEND;
   //    TRECEIVE { S7_SetPoint := 'True'} : TRCV;
   //    TRESET { S7_SetPoint := 'True'} : T_RESET;
   //    TDIAG { S7_SetPoint := 'True'} : T_DIAG;
   //    TDIAG_Status { S7_SetPoint := 'True'} : TDiag_Status;
   //    Blocked_Proc_Timeout : Real;
   //    Rcv_Timeout : Real;
   //    MB_Unit_ID : Byte;
   //    MB_Transaction_ID : Word;
   //    MB_State { ExternalWritable := 'False'} : Word;
   //    SAVED_MB_DATA_ADDR : UDInt;
   //    SAVED_DATA_LEN : UInt;
   //    SAVED_MB_MODE : USInt;
   //    Connection_ID : Word;
   //    Retries : Word;
   //    TEMP_DATA { ExternalWritable := 'False'} : Array[1..263] of Byte;
   //    rcv_timer { ExternalAccessible := 'False'; ExternalVisible := 'False'; ExternalWritable := 'False'; S7_SetPoint := 'True'} : TON_TIME;
   //    wd_timer { ExternalAccessible := 'False'; ExternalVisible := 'False'; ExternalWritable := 'False'; S7_SetPoint := 'True'} : TON_TIME;
   //    Connected : Bool;
   //    Active { ExternalWritable := 'False'} : Bool;
   //    BytesReceived : UDInt;
   // END_VAR
BEGIN
END_DATA_BLOCK

DATA_BLOCK "MbPCS_1-W_slow"   // DB6
// stored: AutoNumber true, DBAccessibleFromOPCUA true, DBAccessibleFromWebserver true, InstanceOfName MB_CLIENT, OfSystemLibElement MB_CLIENT, OfSystemLibVersion 5.2
"MB_CLIENT"
   // VAR_INPUT
   //    REQ : Bool;
   //    DISCONNECT : Bool;
   //    MB_MODE : USInt;
   //    MB_DATA_ADDR : UDInt;
   //    MB_DATA_LEN : UInt;
   // END_VAR
   // VAR_OUTPUT
   //    DONE : Bool;
   //    BUSY : Bool;
   //    ERROR : Bool;
   //    STATUS { ExternalVisible := 'False'} : Word;
   // END_VAR
   // VAR_IN_OUT
   //    MB_DATA_PTR : Variant;
   //    CONNECT : Variant;
   // END_VAR
   // VAR
   //    TCON { S7_SetPoint := 'True'} : TCON;
   //    TDISCON { S7_SetPoint := 'True'} : TDISCON;
   //    TSEND { S7_SetPoint := 'True'} : TSEND;
   //    TRECEIVE { S7_SetPoint := 'True'} : TRCV;
   //    TRESET { S7_SetPoint := 'True'} : T_RESET;
   //    TDIAG { S7_SetPoint := 'True'} : T_DIAG;
   //    TDIAG_Status { S7_SetPoint := 'True'} : TDiag_Status;
   //    Blocked_Proc_Timeout : Real;
   //    Rcv_Timeout : Real;
   //    MB_Unit_ID : Byte;
   //    MB_Transaction_ID : Word;
   //    MB_State { ExternalWritable := 'False'} : Word;
   //    SAVED_MB_DATA_ADDR : UDInt;
   //    SAVED_DATA_LEN : UInt;
   //    SAVED_MB_MODE : USInt;
   //    Connection_ID : Word;
   //    Retries : Word;
   //    TEMP_DATA { ExternalWritable := 'False'} : Array[1..263] of Byte;
   //    rcv_timer { ExternalAccessible := 'False'; ExternalVisible := 'False'; ExternalWritable := 'False'; S7_SetPoint := 'True'} : TON_TIME;
   //    wd_timer { ExternalAccessible := 'False'; ExternalVisible := 'False'; ExternalWritable := 'False'; S7_SetPoint := 'True'} : TON_TIME;
   //    Connected : Bool;
   //    Active { ExternalWritable := 'False'} : Bool;
   //    BytesReceived : UDInt;
   // END_VAR
BEGIN
END_DATA_BLOCK

DATA_BLOCK "MbPCS_2-R_fast"   // DB15
// stored: AutoNumber true, DBAccessibleFromOPCUA true, DBAccessibleFromWebserver true, InstanceOfName MB_CLIENT, OfSystemLibElement MB_CLIENT, OfSystemLibVersion 5.2
"MB_CLIENT"
   // VAR_INPUT
   //    REQ : Bool;
   //    DISCONNECT : Bool;
   //    MB_MODE : USInt;
   //    MB_DATA_ADDR : UDInt;
   //    MB_DATA_LEN : UInt;
   // END_VAR
   // VAR_OUTPUT
   //    DONE : Bool;
   //    BUSY : Bool;
   //    ERROR : Bool;
   //    STATUS { ExternalVisible := 'False'} : Word;
   // END_VAR
   // VAR_IN_OUT
   //    MB_DATA_PTR : Variant;
   //    CONNECT : Variant;
   // END_VAR
   // VAR
   //    TCON { S7_SetPoint := 'True'} : TCON;
   //    TDISCON { S7_SetPoint := 'True'} : TDISCON;
   //    TSEND { S7_SetPoint := 'True'} : TSEND;
   //    TRECEIVE { S7_SetPoint := 'True'} : TRCV;
   //    TRESET { S7_SetPoint := 'True'} : T_RESET;
   //    TDIAG { S7_SetPoint := 'True'} : T_DIAG;
   //    TDIAG_Status { S7_SetPoint := 'True'} : TDiag_Status;
   //    Blocked_Proc_Timeout : Real;
   //    Rcv_Timeout : Real;
   //    MB_Unit_ID : Byte;
   //    MB_Transaction_ID : Word;
   //    MB_State { ExternalWritable := 'False'} : Word;
   //    SAVED_MB_DATA_ADDR : UDInt;
   //    SAVED_DATA_LEN : UInt;
   //    SAVED_MB_MODE : USInt;
   //    Connection_ID : Word;
   //    Retries : Word;
   //    TEMP_DATA { ExternalWritable := 'False'} : Array[1..263] of Byte;
   //    rcv_timer { ExternalAccessible := 'False'; ExternalVisible := 'False'; ExternalWritable := 'False'; S7_SetPoint := 'True'} : TON_TIME;
   //    wd_timer { ExternalAccessible := 'False'; ExternalVisible := 'False'; ExternalWritable := 'False'; S7_SetPoint := 'True'} : TON_TIME;
   //    Connected : Bool;
   //    Active { ExternalWritable := 'False'} : Bool;
   //    BytesReceived : UDInt;
   // END_VAR
BEGIN
END_DATA_BLOCK

DATA_BLOCK "MbPCS_2-R_slow"   // DB14
// stored: AutoNumber true, DBAccessibleFromOPCUA true, DBAccessibleFromWebserver true, InstanceOfName MB_CLIENT, OfSystemLibElement MB_CLIENT, OfSystemLibVersion 5.2
"MB_CLIENT"
   // VAR_INPUT
   //    REQ : Bool;
   //    DISCONNECT : Bool;
   //    MB_MODE : USInt;
   //    MB_DATA_ADDR : UDInt;
   //    MB_DATA_LEN : UInt;
   // END_VAR
   // VAR_OUTPUT
   //    DONE : Bool;
   //    BUSY : Bool;
   //    ERROR : Bool;
   //    STATUS { ExternalVisible := 'False'} : Word;
   // END_VAR
   // VAR_IN_OUT
   //    MB_DATA_PTR : Variant;
   //    CONNECT : Variant;
   // END_VAR
   // VAR
   //    TCON { S7_SetPoint := 'True'} : TCON;
   //    TDISCON { S7_SetPoint := 'True'} : TDISCON;
   //    TSEND { S7_SetPoint := 'True'} : TSEND;
   //    TRECEIVE { S7_SetPoint := 'True'} : TRCV;
   //    TRESET { S7_SetPoint := 'True'} : T_RESET;
   //    TDIAG { S7_SetPoint := 'True'} : T_DIAG;
   //    TDIAG_Status { S7_SetPoint := 'True'} : TDiag_Status;
   //    Blocked_Proc_Timeout : Real;
   //    Rcv_Timeout : Real;
   //    MB_Unit_ID : Byte;
   //    MB_Transaction_ID : Word;
   //    MB_State { ExternalWritable := 'False'} : Word;
   //    SAVED_MB_DATA_ADDR : UDInt;
   //    SAVED_DATA_LEN : UInt;
   //    SAVED_MB_MODE : USInt;
   //    Connection_ID : Word;
   //    Retries : Word;
   //    TEMP_DATA { ExternalWritable := 'False'} : Array[1..263] of Byte;
   //    rcv_timer { ExternalAccessible := 'False'; ExternalVisible := 'False'; ExternalWritable := 'False'; S7_SetPoint := 'True'} : TON_TIME;
   //    wd_timer { ExternalAccessible := 'False'; ExternalVisible := 'False'; ExternalWritable := 'False'; S7_SetPoint := 'True'} : TON_TIME;
   //    Connected : Bool;
   //    Active { ExternalWritable := 'False'} : Bool;
   //    BytesReceived : UDInt;
   // END_VAR
BEGIN
END_DATA_BLOCK

DATA_BLOCK "MbPCS_2-W_fast"   // DB10
// stored: AutoNumber true, DBAccessibleFromOPCUA true, DBAccessibleFromWebserver true, InstanceOfName MB_CLIENT, OfSystemLibElement MB_CLIENT, OfSystemLibVersion 5.2
"MB_CLIENT"
   // VAR_INPUT
   //    REQ : Bool;
   //    DISCONNECT : Bool;
   //    MB_MODE : USInt;
   //    MB_DATA_ADDR : UDInt;
   //    MB_DATA_LEN : UInt;
   // END_VAR
   // VAR_OUTPUT
   //    DONE : Bool;
   //    BUSY : Bool;
   //    ERROR : Bool;
   //    STATUS { ExternalVisible := 'False'} : Word;
   // END_VAR
   // VAR_IN_OUT
   //    MB_DATA_PTR : Variant;
   //    CONNECT : Variant;
   // END_VAR
   // VAR
   //    TCON { S7_SetPoint := 'True'} : TCON;
   //    TDISCON { S7_SetPoint := 'True'} : TDISCON;
   //    TSEND { S7_SetPoint := 'True'} : TSEND;
   //    TRECEIVE { S7_SetPoint := 'True'} : TRCV;
   //    TRESET { S7_SetPoint := 'True'} : T_RESET;
   //    TDIAG { S7_SetPoint := 'True'} : T_DIAG;
   //    TDIAG_Status { S7_SetPoint := 'True'} : TDiag_Status;
   //    Blocked_Proc_Timeout : Real;
   //    Rcv_Timeout : Real;
   //    MB_Unit_ID : Byte;
   //    MB_Transaction_ID : Word;
   //    MB_State { ExternalWritable := 'False'} : Word;
   //    SAVED_MB_DATA_ADDR : UDInt;
   //    SAVED_DATA_LEN : UInt;
   //    SAVED_MB_MODE : USInt;
   //    Connection_ID : Word;
   //    Retries : Word;
   //    TEMP_DATA { ExternalWritable := 'False'} : Array[1..263] of Byte;
   //    rcv_timer { ExternalAccessible := 'False'; ExternalVisible := 'False'; ExternalWritable := 'False'; S7_SetPoint := 'True'} : TON_TIME;
   //    wd_timer { ExternalAccessible := 'False'; ExternalVisible := 'False'; ExternalWritable := 'False'; S7_SetPoint := 'True'} : TON_TIME;
   //    Connected : Bool;
   //    Active { ExternalWritable := 'False'} : Bool;
   //    BytesReceived : UDInt;
   // END_VAR
BEGIN
END_DATA_BLOCK

DATA_BLOCK "MbPCS_2-W_slow"   // DB12
// stored: AutoNumber true, DBAccessibleFromOPCUA true, DBAccessibleFromWebserver true, InstanceOfName MB_CLIENT, OfSystemLibElement MB_CLIENT, OfSystemLibVersion 5.2
"MB_CLIENT"
   // VAR_INPUT
   //    REQ : Bool;
   //    DISCONNECT : Bool;
   //    MB_MODE : USInt;
   //    MB_DATA_ADDR : UDInt;
   //    MB_DATA_LEN : UInt;
   // END_VAR
   // VAR_OUTPUT
   //    DONE : Bool;
   //    BUSY : Bool;
   //    ERROR : Bool;
   //    STATUS { ExternalVisible := 'False'} : Word;
   // END_VAR
   // VAR_IN_OUT
   //    MB_DATA_PTR : Variant;
   //    CONNECT : Variant;
   // END_VAR
   // VAR
   //    TCON { S7_SetPoint := 'True'} : TCON;
   //    TDISCON { S7_SetPoint := 'True'} : TDISCON;
   //    TSEND { S7_SetPoint := 'True'} : TSEND;
   //    TRECEIVE { S7_SetPoint := 'True'} : TRCV;
   //    TRESET { S7_SetPoint := 'True'} : T_RESET;
   //    TDIAG { S7_SetPoint := 'True'} : T_DIAG;
   //    TDIAG_Status { S7_SetPoint := 'True'} : TDiag_Status;
   //    Blocked_Proc_Timeout : Real;
   //    Rcv_Timeout : Real;
   //    MB_Unit_ID : Byte;
   //    MB_Transaction_ID : Word;
   //    MB_State { ExternalWritable := 'False'} : Word;
   //    SAVED_MB_DATA_ADDR : UDInt;
   //    SAVED_DATA_LEN : UInt;
   //    SAVED_MB_MODE : USInt;
   //    Connection_ID : Word;
   //    Retries : Word;
   //    TEMP_DATA { ExternalWritable := 'False'} : Array[1..263] of Byte;
   //    rcv_timer { ExternalAccessible := 'False'; ExternalVisible := 'False'; ExternalWritable := 'False'; S7_SetPoint := 'True'} : TON_TIME;
   //    wd_timer { ExternalAccessible := 'False'; ExternalVisible := 'False'; ExternalWritable := 'False'; S7_SetPoint := 'True'} : TON_TIME;
   //    Connected : Bool;
   //    Active { ExternalWritable := 'False'} : Bool;
   //    BytesReceived : UDInt;
   // END_VAR
BEGIN
END_DATA_BLOCK

DATA_BLOCK "Ton1"   // DB201
{ S7_Optimized_Access := 'TRUE' }
// stored: AutoNumber false, DBAccessibleFromOPCUA true, DBAccessibleFromWebserver true, InstanceOfName IEC_TIMER, OfSystemLibElement IEC_TIMER, OfSystemLibVersion 1.0
"IEC_TIMER"
   // VAR
   //    PT : Time;
   //    ET { ExternalWritable := 'False'} : Time;
   //    IN : Bool;
   //    Q { ExternalWritable := 'False'} : Bool;
   // END_VAR
BEGIN
END_DATA_BLOCK

DATA_BLOCK "LSNTP_Server_DB"   // DB123
VERSION : 2.1
// stored: AutoNumber false, DBAccessibleFromOPCUA true, DBAccessibleFromWebserver true, InstanceOfName LSNTP_Server, InstanceOfType FB
"LSNTP_Server"
   // VAR_INPUT
   //    init : Bool;
   //    referenceId : USInt;
   //    lastTimeSet : DTL;
   //    connID : CONN_OUC;
   //    hwID : HW_ANY;
   // END_VAR
   // VAR_OUTPUT
   //    error : Bool;
   //    statusID : Int;
   //    status : Word;
   // END_VAR
   // VAR
   //    InstTCON { S7_SetPoint := 'True'} : TCON;
   //    InstTURCV { S7_SetPoint := 'True'} : TURCV;
   //    InstTUSEND { S7_SetPoint := 'True'} : TUSEND;
   //    InstTDISCON { S7_SetPoint := 'True'} : TDISCON;
   //    statDiscon : Struct
   //       req : Bool;
   //       done : Bool;
   //       error : Bool;
   //       status : Word;
   //    END_STRUCT;
   //    statCon : Struct
   //       req : Bool;
   //       done : Bool;
   //       error : Bool;
   //       status : Word;
   //       param { S7_SetPoint := 'True'} : TCON_IP_v4;
   //    END_STRUCT;
   //    statRcv : Struct
   //       req : Bool;
   //       busy : Bool;
   //       error : Bool;
   //       ndr : Bool;
   //       len : UDInt;
   //       status : Word;
   //       addr { S7_SetPoint := 'True'} : TADDR_Param;
   //       tel { S7_SetPoint := 'True'} : "LSNTP_typeTelegram";
   //    END_STRUCT;
   //    statSend : Struct
   //       req : Bool;
   //       done : Bool;
   //       reqDone : Bool;
   //       error : Bool;
   //       status : Word;
   //       addr { S7_SetPoint := 'True'} : TADDR_Param;
   //       tel { S7_SetPoint := 'True'} : "LSNTP_typeTelegram";
   //    END_STRUCT;
   //    statState : Int;
   //    statEdge : Struct
   //       init : Bool;
   //    END_STRUCT;
   // END_VAR
BEGIN
END_DATA_BLOCK
